(* IEC 61131-3 sources: AXOpen/src/components.dukane.welders/ctrl/src/Axo_IQ_SeriesWelder (part 3) *)

            array_buffer[128] := TO_BYTE(SHR(TO_DWORD(buf2.PressPostWeld.StaticHoldTime), UINT#24));
            array_buffer[129] := TO_BYTE(SHR(TO_DWORD(buf2.PressPostWeld.StaticHoldTime), UINT#16));
            array_buffer[130] := TO_BYTE(SHR(TO_DWORD(buf2.PressPostWeld.StaticHoldTime),  UINT#8));
            array_buffer[131] := TO_BYTE(     TO_DWORD(buf2.PressPostWeld.StaticHoldTime));

            array_buffer[132] := TO_BYTE(SHR(TO_DWORD(buf2.PressPostWeld.AfterburstAmplitude), UINT#24));
            array_buffer[133] := TO_BYTE(SHR(TO_DWORD(buf2.PressPostWeld.AfterburstAmplitude), UINT#16));
            array_buffer[134] := TO_BYTE(SHR(TO_DWORD(buf2.PressPostWeld.AfterburstAmplitude),  UINT#8));
            array_buffer[135] := TO_BYTE(     TO_DWORD(buf2.PressPostWeld.AfterburstAmplitude));

        END_METHOD

        METHOD PRIVATE buf3_TO_ByteArray
            VAR_IN_OUT
                buf3 : Axo_IQ_SeriesWelder_data3_180bytes;
                array_buffer : ARRAY[0..253] OF BYTE;
            END_VAR

            // ---- TriggerTime.Enable bits → bytes 0..3 ----
            array_buffer[ 0].%X0 := buf3.TriggerTime.Enable._0;
            array_buffer[ 0].%X1 := buf3.TriggerTime.Enable._1;
            array_buffer[ 0].%X2 := buf3.TriggerTime.Enable._2;
            array_buffer[ 0].%X3 := buf3.TriggerTime.Enable._3;
            array_buffer[ 0].%X4 := buf3.TriggerTime.Enable._4;
            array_buffer[ 0].%X5 := buf3.TriggerTime.Enable._5;
            array_buffer[ 0].%X6 := buf3.TriggerTime.Enable._6;
            array_buffer[ 0].%X7 := buf3.TriggerTime.Enable._7;

            array_buffer[ 1].%X0 := buf3.TriggerTime.Enable._8;
            array_buffer[ 1].%X1 := buf3.TriggerTime.Enable._9;
            array_buffer[ 1].%X2 := buf3.TriggerTime.Enable._10;
            array_buffer[ 1].%X3 := buf3.TriggerTime.Enable._11;
            array_buffer[ 1].%X4 := buf3.TriggerTime.Enable._12;
            array_buffer[ 1].%X5 := buf3.TriggerTime.Enable._13;
            array_buffer[ 1].%X6 := buf3.TriggerTime.Enable._14;
            array_buffer[ 1].%X7 := buf3.TriggerTime.Enable._15;

            array_buffer[ 2].%X0 := buf3.TriggerTime.Enable._16;
            array_buffer[ 2].%X1 := buf3.TriggerTime.Enable._17;
            array_buffer[ 2].%X2 := buf3.TriggerTime.Enable._18;
            array_buffer[ 2].%X3 := buf3.TriggerTime.Enable._19;
            array_buffer[ 2].%X4 := buf3.TriggerTime.Enable._20;
            array_buffer[ 2].%X5 := buf3.TriggerTime.Enable._21;
            array_buffer[ 2].%X6 := buf3.TriggerTime.Enable._22;
            array_buffer[ 2].%X7 := buf3.TriggerTime.Enable._23;

            array_buffer[ 3].%X0 := buf3.TriggerTime.Enable.LowerBad_1;
            array_buffer[ 3].%X1 := buf3.TriggerTime.Enable.LowerSuspect_1;
            array_buffer[ 3].%X2 := buf3.TriggerTime.Enable.UpperSuspect_1;
            array_buffer[ 3].%X3 := buf3.TriggerTime.Enable.UpperBad_1;
            array_buffer[ 3].%X4 := buf3.TriggerTime.Enable.Display_1;
            array_buffer[ 3].%X5 := buf3.TriggerTime.Enable._29;
            array_buffer[ 3].%X6 := buf3.TriggerTime.Enable._30;
            array_buffer[ 3].%X7 := buf3.TriggerTime.Enable._31;

            // ---- TriggerTime (DINTs) → bytes 4..19 ----
            array_buffer[ 4] := TO_BYTE(SHR(TO_DWORD(buf3.TriggerTime.LowerBad), UINT#24));
            array_buffer[ 5] := TO_BYTE(SHR(TO_DWORD(buf3.TriggerTime.LowerBad), UINT#16));
            array_buffer[ 6] := TO_BYTE(SHR(TO_DWORD(buf3.TriggerTime.LowerBad),  UINT#8));
            array_buffer[ 7] := TO_BYTE(     TO_DWORD(buf3.TriggerTime.LowerBad));

            array_buffer[ 8] := TO_BYTE(SHR(TO_DWORD(buf3.TriggerTime.LowerSuspect), UINT#24));
            array_buffer[ 9] := TO_BYTE(SHR(TO_DWORD(buf3.TriggerTime.LowerSuspect), UINT#16));
            array_buffer[10] := TO_BYTE(SHR(TO_DWORD(buf3.TriggerTime.LowerSuspect),  UINT#8));
            array_buffer[11] := TO_BYTE(     TO_DWORD(buf3.TriggerTime.LowerSuspect));

            array_buffer[12] := TO_BYTE(SHR(TO_DWORD(buf3.TriggerTime.UpperSuspect), UINT#24));
            array_buffer[13] := TO_BYTE(SHR(TO_DWORD(buf3.TriggerTime.UpperSuspect), UINT#16));
            array_buffer[14] := TO_BYTE(SHR(TO_DWORD(buf3.TriggerTime.UpperSuspect),  UINT#8));
            array_buffer[15] := TO_BYTE(     TO_DWORD(buf3.TriggerTime.UpperSuspect));

            array_buffer[16] := TO_BYTE(SHR(TO_DWORD(buf3.TriggerTime.UpperBad), UINT#24));
            array_buffer[17] := TO_BYTE(SHR(TO_DWORD(buf3.TriggerTime.UpperBad), UINT#16));
            array_buffer[18] := TO_BYTE(SHR(TO_DWORD(buf3.TriggerTime.UpperBad),  UINT#8));
            array_buffer[19] := TO_BYTE(     TO_DWORD(buf3.TriggerTime.UpperBad));

            // ---- TriggerPosition.Enable bits → bytes 20..23 ----
            array_buffer[20].%X0 := buf3.TriggerPosition.Enable._0;
            array_buffer[20].%X1 := buf3.TriggerPosition.Enable._1;
            array_buffer[20].%X2 := buf3.TriggerPosition.Enable._2;
            array_buffer[20].%X3 := buf3.TriggerPosition.Enable._3;
            array_buffer[20].%X4 := buf3.TriggerPosition.Enable._4;
            array_buffer[20].%X5 := buf3.TriggerPosition.Enable._5;
            array_buffer[20].%X6 := buf3.TriggerPosition.Enable._6;
            array_buffer[20].%X7 := buf3.TriggerPosition.Enable._7;

            array_buffer[21].%X0 := buf3.TriggerPosition.Enable._8;
            array_buffer[21].%X1 := buf3.TriggerPosition.Enable._9;
            array_buffer[21].%X2 := buf3.TriggerPosition.Enable._10;
            array_buffer[21].%X3 := buf3.TriggerPosition.Enable._11;
            array_buffer[21].%X4 := buf3.TriggerPosition.Enable._12;
            array_buffer[21].%X5 := buf3.TriggerPosition.Enable._13;
            array_buffer[21].%X6 := buf3.TriggerPosition.Enable._14;
            array_buffer[21].%X7 := buf3.TriggerPosition.Enable._15;

            array_buffer[22].%X0 := buf3.TriggerPosition.Enable._16;
            array_buffer[22].%X1 := buf3.TriggerPosition.Enable._17;
            array_buffer[22].%X2 := buf3.TriggerPosition.Enable._18;
            array_buffer[22].%X3 := buf3.TriggerPosition.Enable._19;
            array_buffer[22].%X4 := buf3.TriggerPosition.Enable._20;
            array_buffer[22].%X5 := buf3.TriggerPosition.Enable._21;
            array_buffer[22].%X6 := buf3.TriggerPosition.Enable._22;
            array_buffer[22].%X7 := buf3.TriggerPosition.Enable._23;

            array_buffer[23].%X0 := buf3.TriggerPosition.Enable.LowerBad_1;
            array_buffer[23].%X1 := buf3.TriggerPosition.Enable.LowerSuspect_1;
            array_buffer[23].%X2 := buf3.TriggerPosition.Enable.UpperSuspect_1;
            array_buffer[23].%X3 := buf3.TriggerPosition.Enable.UpperBad_1;
            array_buffer[23].%X4 := buf3.TriggerPosition.Enable.Display_1;
            array_buffer[23].%X5 := buf3.TriggerPosition.Enable._29;
            array_buffer[23].%X6 := buf3.TriggerPosition.Enable._30;
            array_buffer[23].%X7 := buf3.TriggerPosition.Enable._31;

            // ---- TriggerPosition (DINTs) → bytes 24..39 ----
            array_buffer[24] := TO_BYTE(SHR(TO_DWORD(buf3.TriggerPosition.LowerBad), UINT#24));
            array_buffer[25] := TO_BYTE(SHR(TO_DWORD(buf3.TriggerPosition.LowerBad), UINT#16));
            array_buffer[26] := TO_BYTE(SHR(TO_DWORD(buf3.TriggerPosition.LowerBad),  UINT#8));
            array_buffer[27] := TO_BYTE(     TO_DWORD(buf3.TriggerPosition.LowerBad));

            array_buffer[28] := TO_BYTE(SHR(TO_DWORD(buf3.TriggerPosition.LowerSuspect), UINT#24));
            array_buffer[29] := TO_BYTE(SHR(TO_DWORD(buf3.TriggerPosition.LowerSuspect), UINT#16));
            array_buffer[30] := TO_BYTE(SHR(TO_DWORD(buf3.TriggerPosition.LowerSuspect),  UINT#8));
            array_buffer[31] := TO_BYTE(     TO_DWORD(buf3.TriggerPosition.LowerSuspect));

            array_buffer[32] := TO_BYTE(SHR(TO_DWORD(buf3.TriggerPosition.UpperSuspect), UINT#24));
            array_buffer[33] := TO_BYTE(SHR(TO_DWORD(buf3.TriggerPosition.UpperSuspect), UINT#16));
            array_buffer[34] := TO_BYTE(SHR(TO_DWORD(buf3.TriggerPosition.UpperSuspect),  UINT#8));
            array_buffer[35] := TO_BYTE(     TO_DWORD(buf3.TriggerPosition.UpperSuspect));

            array_buffer[36] := TO_BYTE(SHR(TO_DWORD(buf3.TriggerPosition.UpperBad), UINT#24));
            array_buffer[37] := TO_BYTE(SHR(TO_DWORD(buf3.TriggerPosition.UpperBad), UINT#16));
            array_buffer[38] := TO_BYTE(SHR(TO_DWORD(buf3.TriggerPosition.UpperBad),  UINT#8));
            array_buffer[39] := TO_BYTE(     TO_DWORD(buf3.TriggerPosition.UpperBad));

            // ---- TriggerDelayTime.Enable bits → bytes 40..43 ----
            array_buffer[40].%X0 := buf3.TriggerDelayTime.Enable._0;
            array_buffer[40].%X1 := buf3.TriggerDelayTime.Enable._1;
            array_buffer[40].%X2 := buf3.TriggerDelayTime.Enable._2;
            array_buffer[40].%X3 := buf3.TriggerDelayTime.Enable._3;
            array_buffer[40].%X4 := buf3.TriggerDelayTime.Enable._4;
            array_buffer[40].%X5 := buf3.TriggerDelayTime.Enable._5;
            array_buffer[40].%X6 := buf3.TriggerDelayTime.Enable._6;
            array_buffer[40].%X7 := buf3.TriggerDelayTime.Enable._7;

            array_buffer[41].%X0 := buf3.TriggerDelayTime.Enable._8;
            array_buffer[41].%X1 := buf3.TriggerDelayTime.Enable._9;
            array_buffer[41].%X2 := buf3.TriggerDelayTime.Enable._10;
            array_buffer[41].%X3 := buf3.TriggerDelayTime.Enable._11;
            array_buffer[41].%X4 := buf3.TriggerDelayTime.Enable._12;
            array_buffer[41].%X5 := buf3.TriggerDelayTime.Enable._13;
            array_buffer[41].%X6 := buf3.TriggerDelayTime.Enable._14;
            array_buffer[41].%X7 := buf3.TriggerDelayTime.Enable._15;

            array_buffer[42].%X0 := buf3.TriggerDelayTime.Enable._16;
            array_buffer[42].%X1 := buf3.TriggerDelayTime.Enable._17;
            array_buffer[42].%X2 := buf3.TriggerDelayTime.Enable._18;
            array_buffer[42].%X3 := buf3.TriggerDelayTime.Enable._19;
            array_buffer[42].%X4 := buf3.TriggerDelayTime.Enable._20;
            array_buffer[42].%X5 := buf3.TriggerDelayTime.Enable._21;
            array_buffer[42].%X6 := buf3.TriggerDelayTime.Enable._22;
            array_buffer[42].%X7 := buf3.TriggerDelayTime.Enable._23;

            array_buffer[43].%X0 := buf3.TriggerDelayTime.Enable.LowerBad_1;
            array_buffer[43].%X1 := buf3.TriggerDelayTime.Enable.LowerSuspect_1;
            array_buffer[43].%X2 := buf3.TriggerDelayTime.Enable.UpperSuspect_1;
            array_buffer[43].%X3 := buf3.TriggerDelayTime.Enable.UpperBad_1;
            array_buffer[43].%X4 := buf3.TriggerDelayTime.Enable.Display_1;
            array_buffer[43].%X5 := buf3.TriggerDelayTime.Enable._29;
            array_buffer[43].%X6 := buf3.TriggerDelayTime.Enable._30;
            array_buffer[43].%X7 := buf3.TriggerDelayTime.Enable._31;

            // ---- TriggerDelayTime (DINTs) → bytes 44..59 ----
            array_buffer[44] := TO_BYTE(SHR(TO_DWORD(buf3.TriggerDelayTime.LowerBad), UINT#24));
            array_buffer[45] := TO_BYTE(SHR(TO_DWORD(buf3.TriggerDelayTime.LowerBad), UINT#16));
            array_buffer[46] := TO_BYTE(SHR(TO_DWORD(buf3.TriggerDelayTime.LowerBad),  UINT#8));
            array_buffer[47] := TO_BYTE(     TO_DWORD(buf3.TriggerDelayTime.LowerBad));

            array_buffer[48] := TO_BYTE(SHR(TO_DWORD(buf3.TriggerDelayTime.LowerSuspect), UINT#24));
            array_buffer[49] := TO_BYTE(SHR(TO_DWORD(buf3.TriggerDelayTime.LowerSuspect), UINT#16));
            array_buffer[50] := TO_BYTE(SHR(TO_DWORD(buf3.TriggerDelayTime.LowerSuspect),  UINT#8));
            array_buffer[51] := TO_BYTE(     TO_DWORD(buf3.TriggerDelayTime.LowerSuspect));

            array_buffer[52] := TO_BYTE(SHR(TO_DWORD(buf3.TriggerDelayTime.UpperSuspect), UINT#24));
            array_buffer[53] := TO_BYTE(SHR(TO_DWORD(buf3.TriggerDelayTime.UpperSuspect), UINT#16));
            array_buffer[54] := TO_BYTE(SHR(TO_DWORD(buf3.TriggerDelayTime.UpperSuspect),  UINT#8));
            array_buffer[55] := TO_BYTE(     TO_DWORD(buf3.TriggerDelayTime.UpperSuspect));

            array_buffer[56] := TO_BYTE(SHR(TO_DWORD(buf3.TriggerDelayTime.UpperBad), UINT#24));
            array_buffer[57] := TO_BYTE(SHR(TO_DWORD(buf3.TriggerDelayTime.UpperBad), UINT#16));
            array_buffer[58] := TO_BYTE(SHR(TO_DWORD(buf3.TriggerDelayTime.UpperBad),  UINT#8));
            array_buffer[59] := TO_BYTE(     TO_DWORD(buf3.TriggerDelayTime.UpperBad));

            // ---- TriggerDelayDistance.Enable bits → bytes 60..63 ----
            array_buffer[60].%X0 := buf3.TriggerDelayDistance.Enable._0;
            array_buffer[60].%X1 := buf3.TriggerDelayDistance.Enable._1;
            array_buffer[60].%X2 := buf3.TriggerDelayDistance.Enable._2;
            array_buffer[60].%X3 := buf3.TriggerDelayDistance.Enable._3;
            array_buffer[60].%X4 := buf3.TriggerDelayDistance.Enable._4;
            array_buffer[60].%X5 := buf3.TriggerDelayDistance.Enable._5;
            array_buffer[60].%X6 := buf3.TriggerDelayDistance.Enable._6;
            array_buffer[60].%X7 := buf3.TriggerDelayDistance.Enable._7;

            array_buffer[61].%X0 := buf3.TriggerDelayDistance.Enable._8;
            array_buffer[61].%X1 := buf3.TriggerDelayDistance.Enable._9;
            array_buffer[61].%X2 := buf3.TriggerDelayDistance.Enable._10;
            array_buffer[61].%X3 := buf3.TriggerDelayDistance.Enable._11;
            array_buffer[61].%X4 := buf3.TriggerDelayDistance.Enable._12;
            array_buffer[61].%X5 := buf3.TriggerDelayDistance.Enable._13;
            array_buffer[61].%X6 := buf3.TriggerDelayDistance.Enable._14;
            array_buffer[61].%X7 := buf3.TriggerDelayDistance.Enable._15;

            array_buffer[62].%X0 := buf3.TriggerDelayDistance.Enable._16;
            array_buffer[62].%X1 := buf3.TriggerDelayDistance.Enable._17;
            array_buffer[62].%X2 := buf3.TriggerDelayDistance.Enable._18;
            array_buffer[62].%X3 := buf3.TriggerDelayDistance.Enable._19;
            array_buffer[62].%X4 := buf3.TriggerDelayDistance.Enable._20;
            array_buffer[62].%X5 := buf3.TriggerDelayDistance.Enable._21;
            array_buffer[62].%X6 := buf3.TriggerDelayDistance.Enable._22;
            array_buffer[62].%X7 := buf3.TriggerDelayDistance.Enable._23;

            array_buffer[63].%X0 := buf3.TriggerDelayDistance.Enable.LowerBad_1;
            array_buffer[63].%X1 := buf3.TriggerDelayDistance.Enable.LowerSuspect_1;
            array_buffer[63].%X2 := buf3.TriggerDelayDistance.Enable.UpperSuspect_1;
            array_buffer[63].%X3 := buf3.TriggerDelayDistance.Enable.UpperBad_1;
            array_buffer[63].%X4 := buf3.TriggerDelayDistance.Enable.Display_1;
            array_buffer[63].%X5 := buf3.TriggerDelayDistance.Enable._29;
            array_buffer[63].%X6 := buf3.TriggerDelayDistance.Enable._30;
            array_buffer[63].%X7 := buf3.TriggerDelayDistance.Enable._31;

            // ---- TriggerDelayDistance (DINTs) → bytes 64..79 ----
            array_buffer[64] := TO_BYTE(SHR(TO_DWORD(buf3.TriggerDelayDistance.LowerBad), UINT#24));
            array_buffer[65] := TO_BYTE(SHR(TO_DWORD(buf3.TriggerDelayDistance.LowerBad), UINT#16));
            array_buffer[66] := TO_BYTE(SHR(TO_DWORD(buf3.TriggerDelayDistance.LowerBad),  UINT#8));
            array_buffer[67] := TO_BYTE(     TO_DWORD(buf3.TriggerDelayDistance.LowerBad));

            array_buffer[68] := TO_BYTE(SHR(TO_DWORD(buf3.TriggerDelayDistance.LowerSuspect), UINT#24));
            array_buffer[69] := TO_BYTE(SHR(TO_DWORD(buf3.TriggerDelayDistance.LowerSuspect), UINT#16));
            array_buffer[70] := TO_BYTE(SHR(TO_DWORD(buf3.TriggerDelayDistance.LowerSuspect),  UINT#8));
            array_buffer[71] := TO_BYTE(     TO_DWORD(buf3.TriggerDelayDistance.LowerSuspect));

            array_buffer[72] := TO_BYTE(SHR(TO_DWORD(buf3.TriggerDelayDistance.UpperSuspect), UINT#24));
            array_buffer[73] := TO_BYTE(SHR(TO_DWORD(buf3.TriggerDelayDistance.UpperSuspect), UINT#16));
            array_buffer[74] := TO_BYTE(SHR(TO_DWORD(buf3.TriggerDelayDistance.UpperSuspect),  UINT#8));
            array_buffer[75] := TO_BYTE(     TO_DWORD(buf3.TriggerDelayDistance.UpperSuspect));

            array_buffer[76] := TO_BYTE(SHR(TO_DWORD(buf3.TriggerDelayDistance.UpperBad), UINT#24));
            array_buffer[77] := TO_BYTE(SHR(TO_DWORD(buf3.TriggerDelayDistance.UpperBad), UINT#16));
            array_buffer[78] := TO_BYTE(SHR(TO_DWORD(buf3.TriggerDelayDistance.UpperBad),  UINT#8));
            array_buffer[79] := TO_BYTE(     TO_DWORD(buf3.TriggerDelayDistance.UpperBad));

            // ---- Weld1Distance.Enable bits → bytes 80..83 ----
            array_buffer[80].%X0 := buf3.Weld1Distance.Enable._0;
            array_buffer[80].%X1 := buf3.Weld1Distance.Enable._1;
            array_buffer[80].%X2 := buf3.Weld1Distance.Enable._2;
            array_buffer[80].%X3 := buf3.Weld1Distance.Enable._3;
            array_buffer[80].%X4 := buf3.Weld1Distance.Enable._4;
            array_buffer[80].%X5 := buf3.Weld1Distance.Enable._5;
            array_buffer[80].%X6 := buf3.Weld1Distance.Enable._6;
            array_buffer[80].%X7 := buf3.Weld1Distance.Enable._7;

            array_buffer[81].%X0 := buf3.Weld1Distance.Enable._8;
            array_buffer[81].%X1 := buf3.Weld1Distance.Enable._9;
            array_buffer[81].%X2 := buf3.Weld1Distance.Enable._10;
            array_buffer[81].%X3 := buf3.Weld1Distance.Enable._11;
            array_buffer[81].%X4 := buf3.Weld1Distance.Enable._12;
            array_buffer[81].%X5 := buf3.Weld1Distance.Enable._13;
            array_buffer[81].%X6 := buf3.Weld1Distance.Enable._14;
            array_buffer[81].%X7 := buf3.Weld1Distance.Enable._15;

            array_buffer[82].%X0 := buf3.Weld1Distance.Enable._16;
            array_buffer[82].%X1 := buf3.Weld1Distance.Enable._17;
            array_buffer[82].%X2 := buf3.Weld1Distance.Enable._18;
            array_buffer[82].%X3 := buf3.Weld1Distance.Enable._19;
            array_buffer[82].%X4 := buf3.Weld1Distance.Enable._20;
            array_buffer[82].%X5 := buf3.Weld1Distance.Enable._21;
            array_buffer[82].%X6 := buf3.Weld1Distance.Enable._22;
            array_buffer[82].%X7 := buf3.Weld1Distance.Enable._23;

            array_buffer[83].%X0 := buf3.Weld1Distance.Enable.LowerBad_1;
            array_buffer[83].%X1 := buf3.Weld1Distance.Enable.LowerSuspect_1;
            array_buffer[83].%X2 := buf3.Weld1Distance.Enable.UpperSuspect_1;
            array_buffer[83].%X3 := buf3.Weld1Distance.Enable.UpperBad_1;
            array_buffer[83].%X4 := buf3.Weld1Distance.Enable.Display_1;
            array_buffer[83].%X5 := buf3.Weld1Distance.Enable._29;
            array_buffer[83].%X6 := buf3.Weld1Distance.Enable._30;
            array_buffer[83].%X7 := buf3.Weld1Distance.Enable._31;

            // ---- Weld1Distance (DINTs) → bytes 84..99 ----
            array_buffer[84] := TO_BYTE(SHR(TO_DWORD(buf3.Weld1Distance.LowerBad), UINT#24));
            array_buffer[85] := TO_BYTE(SHR(TO_DWORD(buf3.Weld1Distance.LowerBad), UINT#16));
            array_buffer[86] := TO_BYTE(SHR(TO_DWORD(buf3.Weld1Distance.LowerBad),  UINT#8));
            array_buffer[87] := TO_BYTE(     TO_DWORD(buf3.Weld1Distance.LowerBad));

            array_buffer[88] := TO_BYTE(SHR(TO_DWORD(buf3.Weld1Distance.LowerSuspect), UINT#24));
            array_buffer[89] := TO_BYTE(SHR(TO_DWORD(buf3.Weld1Distance.LowerSuspect), UINT#16));
            array_buffer[90] := TO_BYTE(SHR(TO_DWORD(buf3.Weld1Distance.LowerSuspect),  UINT#8));
            array_buffer[91] := TO_BYTE(     TO_DWORD(buf3.Weld1Distance.LowerSuspect));

            array_buffer[92] := TO_BYTE(SHR(TO_DWORD(buf3.Weld1Distance.UpperSuspect), UINT#24));
            array_buffer[93] := TO_BYTE(SHR(TO_DWORD(buf3.Weld1Distance.UpperSuspect), UINT#16));
            array_buffer[94] := TO_BYTE(SHR(TO_DWORD(buf3.Weld1Distance.UpperSuspect),  UINT#8));
            array_buffer[95] := TO_BYTE(     TO_DWORD(buf3.Weld1Distance.UpperSuspect));

            array_buffer[96] := TO_BYTE(SHR(TO_DWORD(buf3.Weld1Distance.UpperBad), UINT#24));
            array_buffer[97] := TO_BYTE(SHR(TO_DWORD(buf3.Weld1Distance.UpperBad), UINT#16));
            array_buffer[98] := TO_BYTE(SHR(TO_DWORD(buf3.Weld1Distance.UpperBad),  UINT#8));
            array_buffer[99] := TO_BYTE(     TO_DWORD(buf3.Weld1Distance.UpperBad));

            // ---- Weld1Position.Enable bits → bytes 100..103 ----
            array_buffer[100].%X0 := buf3.Weld1Position.Enable._0;
            array_buffer[100].%X1 := buf3.Weld1Position.Enable._1;
            array_buffer[100].%X2 := buf3.Weld1Position.Enable._2;
            array_buffer[100].%X3 := buf3.Weld1Position.Enable._3;
            array_buffer[100].%X4 := buf3.Weld1Position.Enable._4;
            array_buffer[100].%X5 := buf3.Weld1Position.Enable._5;
            array_buffer[100].%X6 := buf3.Weld1Position.Enable._6;
            array_buffer[100].%X7 := buf3.Weld1Position.Enable._7;

            array_buffer[101].%X0 := buf3.Weld1Position.Enable._8;
            array_buffer[101].%X1 := buf3.Weld1Position.Enable._9;
            array_buffer[101].%X2 := buf3.Weld1Position.Enable._10;
            array_buffer[101].%X3 := buf3.Weld1Position.Enable._11;
            array_buffer[101].%X4 := buf3.Weld1Position.Enable._12;
            array_buffer[101].%X5 := buf3.Weld1Position.Enable._13;
            array_buffer[101].%X6 := buf3.Weld1Position.Enable._14;
            array_buffer[101].%X7 := buf3.Weld1Position.Enable._15;

            array_buffer[102].%X0 := buf3.Weld1Position.Enable._16;
            array_buffer[102].%X1 := buf3.Weld1Position.Enable._17;
            array_buffer[102].%X2 := buf3.Weld1Position.Enable._18;
            array_buffer[102].%X3 := buf3.Weld1Position.Enable._19;
            array_buffer[102].%X4 := buf3.Weld1Position.Enable._20;
            array_buffer[102].%X5 := buf3.Weld1Position.Enable._21;
            array_buffer[102].%X6 := buf3.Weld1Position.Enable._22;
            array_buffer[102].%X7 := buf3.Weld1Position.Enable._23;

            array_buffer[103].%X0 := buf3.Weld1Position.Enable.LowerBad_1;
            array_buffer[103].%X1 := buf3.Weld1Position.Enable.LowerSuspect_1;
            array_buffer[103].%X2 := buf3.Weld1Position.Enable.UpperSuspect_1;
            array_buffer[103].%X3 := buf3.Weld1Position.Enable.UpperBad_1;
            array_buffer[103].%X4 := buf3.Weld1Position.Enable.Display_1;
            array_buffer[103].%X5 := buf3.Weld1Position.Enable._29;
            array_buffer[103].%X6 := buf3.Weld1Position.Enable._30;
            array_buffer[103].%X7 := buf3.Weld1Position.Enable._31;

            // ---- Weld1Position (DINTs) → bytes 104..119 ----
            array_buffer[104] := TO_BYTE(SHR(TO_DWORD(buf3.Weld1Position.LowerBad), UINT#24));
            array_buffer[105] := TO_BYTE(SHR(TO_DWORD(buf3.Weld1Position.LowerBad), UINT#16));
            array_buffer[106] := TO_BYTE(SHR(TO_DWORD(buf3.Weld1Position.LowerBad),  UINT#8));
            array_buffer[107] := TO_BYTE(     TO_DWORD(buf3.Weld1Position.LowerBad));

            array_buffer[108] := TO_BYTE(SHR(TO_DWORD(buf3.Weld1Position.LowerSuspect), UINT#24));
            array_buffer[109] := TO_BYTE(SHR(TO_DWORD(buf3.Weld1Position.LowerSuspect), UINT#16));
            array_buffer[110] := TO_BYTE(SHR(TO_DWORD(buf3.Weld1Position.LowerSuspect),  UINT#8));
            array_buffer[111] := TO_BYTE(     TO_DWORD(buf3.Weld1Position.LowerSuspect));

            array_buffer[112] := TO_BYTE(SHR(TO_DWORD(buf3.Weld1Position.UpperSuspect), UINT#24));
            array_buffer[113] := TO_BYTE(SHR(TO_DWORD(buf3.Weld1Position.UpperSuspect), UINT#16));
            array_buffer[114] := TO_BYTE(SHR(TO_DWORD(buf3.Weld1Position.UpperSuspect),  UINT#8));
            array_buffer[115] := TO_BYTE(     TO_DWORD(buf3.Weld1Position.UpperSuspect));

            array_buffer[116] := TO_BYTE(SHR(TO_DWORD(buf3.Weld1Position.UpperBad), UINT#24));
            array_buffer[117] := TO_BYTE(SHR(TO_DWORD(buf3.Weld1Position.UpperBad), UINT#16));
            array_buffer[118] := TO_BYTE(SHR(TO_DWORD(buf3.Weld1Position.UpperBad),  UINT#8));
            array_buffer[119] := TO_BYTE(     TO_DWORD(buf3.Weld1Position.UpperBad));

            // ---- Weld2Time.Enable bits → bytes 120..123 ----
            array_buffer[120].%X0 := buf3.Weld2Time.Enable._0;
            array_buffer[120].%X1 := buf3.Weld2Time.Enable._1;
            array_buffer[120].%X2 := buf3.Weld2Time.Enable._2;
            array_buffer[120].%X3 := buf3.Weld2Time.Enable._3;
            array_buffer[120].%X4 := buf3.Weld2Time.Enable._4;
            array_buffer[120].%X5 := buf3.Weld2Time.Enable._5;
            array_buffer[120].%X6 := buf3.Weld2Time.Enable._6;
            array_buffer[120].%X7 := buf3.Weld2Time.Enable._7;

            array_buffer[121].%X0 := buf3.Weld2Time.Enable._8;
            array_buffer[121].%X1 := buf3.Weld2Time.Enable._9;
            array_buffer[121].%X2 := buf3.Weld2Time.Enable._10;
            array_buffer[121].%X3 := buf3.Weld2Time.Enable._11;
            array_buffer[121].%X4 := buf3.Weld2Time.Enable._12;
            array_buffer[121].%X5 := buf3.Weld2Time.Enable._13;
            array_buffer[121].%X6 := buf3.Weld2Time.Enable._14;
            array_buffer[121].%X7 := buf3.Weld2Time.Enable._15;

            array_buffer[122].%X0 := buf3.Weld2Time.Enable._16;
            array_buffer[122].%X1 := buf3.Weld2Time.Enable._17;
            array_buffer[122].%X2 := buf3.Weld2Time.Enable._18;
            array_buffer[122].%X3 := buf3.Weld2Time.Enable._19;
            array_buffer[122].%X4 := buf3.Weld2Time.Enable._20;
            array_buffer[122].%X5 := buf3.Weld2Time.Enable._21;
            array_buffer[122].%X6 := buf3.Weld2Time.Enable._22;
            array_buffer[122].%X7 := buf3.Weld2Time.Enable._23;

            array_buffer[123].%X0 := buf3.Weld2Time.Enable.LowerBad_1;
            array_buffer[123].%X1 := buf3.Weld2Time.Enable.LowerSuspect_1;
            array_buffer[123].%X2 := buf3.Weld2Time.Enable.UpperSuspect_1;
            array_buffer[123].%X3 := buf3.Weld2Time.Enable.UpperBad_1;
            array_buffer[123].%X4 := buf3.Weld2Time.Enable.Display_1;
            array_buffer[123].%X5 := buf3.Weld2Time.Enable._29;
            array_buffer[123].%X6 := buf3.Weld2Time.Enable._30;
            array_buffer[123].%X7 := buf3.Weld2Time.Enable._31;

            // ---- Weld2Time (DINTs) → bytes 124..139 ----
            array_buffer[124] := TO_BYTE(SHR(TO_DWORD(buf3.Weld2Time.LowerBad), UINT#24));
            array_buffer[125] := TO_BYTE(SHR(TO_DWORD(buf3.Weld2Time.LowerBad), UINT#16));
            array_buffer[126] := TO_BYTE(SHR(TO_DWORD(buf3.Weld2Time.LowerBad),  UINT#8));
            array_buffer[127] := TO_BYTE(     TO_DWORD(buf3.Weld2Time.LowerBad));

            array_buffer[128] := TO_BYTE(SHR(TO_DWORD(buf3.Weld2Time.LowerSuspect), UINT#24));
            array_buffer[129] := TO_BYTE(SHR(TO_DWORD(buf3.Weld2Time.LowerSuspect), UINT#16));
            array_buffer[130] := TO_BYTE(SHR(TO_DWORD(buf3.Weld2Time.LowerSuspect),  UINT#8));
            array_buffer[131] := TO_BYTE(     TO_DWORD(buf3.Weld2Time.LowerSuspect));

            array_buffer[132] := TO_BYTE(SHR(TO_DWORD(buf3.Weld2Time.UpperSuspect), UINT#24));
            array_buffer[133] := TO_BYTE(SHR(TO_DWORD(buf3.Weld2Time.UpperSuspect), UINT#16));
            array_buffer[134] := TO_BYTE(SHR(TO_DWORD(buf3.Weld2Time.UpperSuspect),  UINT#8));
            array_buffer[135] := TO_BYTE(     TO_DWORD(buf3.Weld2Time.UpperSuspect));

            array_buffer[136] := TO_BYTE(SHR(TO_DWORD(buf3.Weld2Time.UpperBad), UINT#24));
            array_buffer[137] := TO_BYTE(SHR(TO_DWORD(buf3.Weld2Time.UpperBad), UINT#16));
            array_buffer[138] := TO_BYTE(SHR(TO_DWORD(buf3.Weld2Time.UpperBad),  UINT#8));
            array_buffer[139] := TO_BYTE(     TO_DWORD(buf3.Weld2Time.UpperBad));

            // ---- Weld2Energy.Enable bits → bytes 140..143 ----
            array_buffer[140].%X0 := buf3.Weld2Energy.Enable._0;
            array_buffer[140].%X1 := buf3.Weld2Energy.Enable._1;
            array_buffer[140].%X2 := buf3.Weld2Energy.Enable._2;
            array_buffer[140].%X3 := buf3.Weld2Energy.Enable._3;
            array_buffer[140].%X4 := buf3.Weld2Energy.Enable._4;
            array_buffer[140].%X5 := buf3.Weld2Energy.Enable._5;
            array_buffer[140].%X6 := buf3.Weld2Energy.Enable._6;
            array_buffer[140].%X7 := buf3.Weld2Energy.Enable._7;

            array_buffer[141].%X0 := buf3.Weld2Energy.Enable._8;
            array_buffer[141].%X1 := buf3.Weld2Energy.Enable._9;
            array_buffer[141].%X2 := buf3.Weld2Energy.Enable._10;
            array_buffer[141].%X3 := buf3.Weld2Energy.Enable._11;
            array_buffer[141].%X4 := buf3.Weld2Energy.Enable._12;
            array_buffer[141].%X5 := buf3.Weld2Energy.Enable._13;
            array_buffer[141].%X6 := buf3.Weld2Energy.Enable._14;
            array_buffer[141].%X7 := buf3.Weld2Energy.Enable._15;

            array_buffer[142].%X0 := buf3.Weld2Energy.Enable._16;
            array_buffer[142].%X1 := buf3.Weld2Energy.Enable._17;
            array_buffer[142].%X2 := buf3.Weld2Energy.Enable._18;
            array_buffer[142].%X3 := buf3.Weld2Energy.Enable._19;
            array_buffer[142].%X4 := buf3.Weld2Energy.Enable._20;
            array_buffer[142].%X5 := buf3.Weld2Energy.Enable._21;
            array_buffer[142].%X6 := buf3.Weld2Energy.Enable._22;
            array_buffer[142].%X7 := buf3.Weld2Energy.Enable._23;

            array_buffer[143].%X0 := buf3.Weld2Energy.Enable.LowerBad_1;
            array_buffer[143].%X1 := buf3.Weld2Energy.Enable.LowerSuspect_1;
            array_buffer[143].%X2 := buf3.Weld2Energy.Enable.UpperSuspect_1;
            array_buffer[143].%X3 := buf3.Weld2Energy.Enable.UpperBad_1;
            array_buffer[143].%X4 := buf3.Weld2Energy.Enable.Display_1;
            array_buffer[143].%X5 := buf3.Weld2Energy.Enable._29;
            array_buffer[143].%X6 := buf3.Weld2Energy.Enable._30;
            array_buffer[143].%X7 := buf3.Weld2Energy.Enable._31;

            // ---- Weld2Energy (DINTs) → bytes 144..159 ----
            array_buffer[144] := TO_BYTE(SHR(TO_DWORD(buf3.Weld2Energy.LowerBad), UINT#24));
            array_buffer[145] := TO_BYTE(SHR(TO_DWORD(buf3.Weld2Energy.LowerBad), UINT#16));
            array_buffer[146] := TO_BYTE(SHR(TO_DWORD(buf3.Weld2Energy.LowerBad),  UINT#8));
            array_buffer[147] := TO_BYTE(     TO_DWORD(buf3.Weld2Energy.LowerBad));

            array_buffer[148] := TO_BYTE(SHR(TO_DWORD(buf3.Weld2Energy.LowerSuspect), UINT#24));
            array_buffer[149] := TO_BYTE(SHR(TO_DWORD(buf3.Weld2Energy.LowerSuspect), UINT#16));
            array_buffer[150] := TO_BYTE(SHR(TO_DWORD(buf3.Weld2Energy.LowerSuspect),  UINT#8));
            array_buffer[151] := TO_BYTE(     TO_DWORD(buf3.Weld2Energy.LowerSuspect));

            array_buffer[152] := TO_BYTE(SHR(TO_DWORD(buf3.Weld2Energy.UpperSuspect), UINT#24));
            array_buffer[153] := TO_BYTE(SHR(TO_DWORD(buf3.Weld2Energy.UpperSuspect), UINT#16));
            array_buffer[154] := TO_BYTE(SHR(TO_DWORD(buf3.Weld2Energy.UpperSuspect),  UINT#8));
            array_buffer[155] := TO_BYTE(     TO_DWORD(buf3.Weld2Energy.UpperSuspect));

            array_buffer[156] := TO_BYTE(SHR(TO_DWORD(buf3.Weld2Energy.UpperBad), UINT#24));
            array_buffer[157] := TO_BYTE(SHR(TO_DWORD(buf3.Weld2Energy.UpperBad), UINT#16));
            array_buffer[158] := TO_BYTE(SHR(TO_DWORD(buf3.Weld2Energy.UpperBad),  UINT#8));
            array_buffer[159] := TO_BYTE(     TO_DWORD(buf3.Weld2Energy.UpperBad));

            // ---- Weld2Power.Enable bits → bytes 160..163 ----
            array_buffer[160].%X0 := buf3.Weld2Power.Enable._0;
            array_buffer[160].%X1 := buf3.Weld2Power.Enable._1;
            array_buffer[160].%X2 := buf3.Weld2Power.Enable._2;
            array_buffer[160].%X3 := buf3.Weld2Power.Enable._3;
            array_buffer[160].%X4 := buf3.Weld2Power.Enable._4;
            array_buffer[160].%X5 := buf3.Weld2Power.Enable._5;
            array_buffer[160].%X6 := buf3.Weld2Power.Enable._6;
            array_buffer[160].%X7 := buf3.Weld2Power.Enable._7;

            array_buffer[161].%X0 := buf3.Weld2Power.Enable._8;
            array_buffer[161].%X1 := buf3.Weld2Power.Enable._9;
            array_buffer[161].%X2 := buf3.Weld2Power.Enable._10;
            array_buffer[161].%X3 := buf3.Weld2Power.Enable._11;
            array_buffer[161].%X4 := buf3.Weld2Power.Enable._12;
            array_buffer[161].%X5 := buf3.Weld2Power.Enable._13;
            array_buffer[161].%X6 := buf3.Weld2Power.Enable._14;
            array_buffer[161].%X7 := buf3.Weld2Power.Enable._15;

            array_buffer[162].%X0 := buf3.Weld2Power.Enable._16;
            array_buffer[162].%X1 := buf3.Weld2Power.Enable._17;
            array_buffer[162].%X2 := buf3.Weld2Power.Enable._18;
            array_buffer[162].%X3 := buf3.Weld2Power.Enable._19;
            array_buffer[162].%X4 := buf3.Weld2Power.Enable._20;
            array_buffer[162].%X5 := buf3.Weld2Power.Enable._21;
            array_buffer[162].%X6 := buf3.Weld2Power.Enable._22;
            array_buffer[162].%X7 := buf3.Weld2Power.Enable._23;

            array_buffer[163].%X0 := buf3.Weld2Power.Enable.LowerBad_1;
            array_buffer[163].%X1 := buf3.Weld2Power.Enable.LowerSuspect_1;
            array_buffer[163].%X2 := buf3.Weld2Power.Enable.UpperSuspect_1;
            array_buffer[163].%X3 := buf3.Weld2Power.Enable.UpperBad_1;
            array_buffer[163].%X4 := buf3.Weld2Power.Enable.Display_1;
            array_buffer[163].%X5 := buf3.Weld2Power.Enable._29;
            array_buffer[163].%X6 := buf3.Weld2Power.Enable._30;
            array_buffer[163].%X7 := buf3.Weld2Power.Enable._31;

            // ---- Weld2Power (DINTs) → bytes 164..179 ----
            array_buffer[164] := TO_BYTE(SHR(TO_DWORD(buf3.Weld2Power.LowerBad), UINT#24));
            array_buffer[165] := TO_BYTE(SHR(TO_DWORD(buf3.Weld2Power.LowerBad), UINT#16));
            array_buffer[166] := TO_BYTE(SHR(TO_DWORD(buf3.Weld2Power.LowerBad),  UINT#8));
            array_buffer[167] := TO_BYTE(     TO_DWORD(buf3.Weld2Power.LowerBad));

            array_buffer[168] := TO_BYTE(SHR(TO_DWORD(buf3.Weld2Power.LowerSuspect), UINT#24));
            array_buffer[169] := TO_BYTE(SHR(TO_DWORD(buf3.Weld2Power.LowerSuspect), UINT#16));
            array_buffer[170] := TO_BYTE(SHR(TO_DWORD(buf3.Weld2Power.LowerSuspect),  UINT#8));
            array_buffer[171] := TO_BYTE(     TO_DWORD(buf3.Weld2Power.LowerSuspect));

            array_buffer[172] := TO_BYTE(SHR(TO_DWORD(buf3.Weld2Power.UpperSuspect), UINT#24));
            array_buffer[173] := TO_BYTE(SHR(TO_DWORD(buf3.Weld2Power.UpperSuspect), UINT#16));
            array_buffer[174] := TO_BYTE(SHR(TO_DWORD(buf3.Weld2Power.UpperSuspect),  UINT#8));
            array_buffer[175] := TO_BYTE(     TO_DWORD(buf3.Weld2Power.UpperSuspect));

            array_buffer[176] := TO_BYTE(SHR(TO_DWORD(buf3.Weld2Power.UpperBad), UINT#24));
            array_buffer[177] := TO_BYTE(SHR(TO_DWORD(buf3.Weld2Power.UpperBad), UINT#16));
            array_buffer[178] := TO_BYTE(SHR(TO_DWORD(buf3.Weld2Power.UpperBad),  UINT#8));
            array_buffer[179] := TO_BYTE(     TO_DWORD(buf3.Weld2Power.UpperBad));

        END_METHOD

        METHOD PRIVATE buf4_TO_ByteArray
            VAR_IN_OUT
                buf4 : Axo_IQ_SeriesWelder_data4_200bytes;
                array_buffer : ARRAY[0..253] OF BYTE;
            END_VAR

            // ---- Weld2Distance.Enable bits → bytes 0..3 ----
            array_buffer[ 0].%X0 := buf4.Weld2Distance.Enable._0;
            array_buffer[ 0].%X1 := buf4.Weld2Distance.Enable._1;
            array_buffer[ 0].%X2 := buf4.Weld2Distance.Enable._2;
            array_buffer[ 0].%X3 := buf4.Weld2Distance.Enable._3;
            array_buffer[ 0].%X4 := buf4.Weld2Distance.Enable._4;
            array_buffer[ 0].%X5 := buf4.Weld2Distance.Enable._5;
            array_buffer[ 0].%X6 := buf4.Weld2Distance.Enable._6;
            array_buffer[ 0].%X7 := buf4.Weld2Distance.Enable._7;

            array_buffer[ 1].%X0 := buf4.Weld2Distance.Enable._8;
            array_buffer[ 1].%X1 := buf4.Weld2Distance.Enable._9;
            array_buffer[ 1].%X2 := buf4.Weld2Distance.Enable._10;
            array_buffer[ 1].%X3 := buf4.Weld2Distance.Enable._11;
            array_buffer[ 1].%X4 := buf4.Weld2Distance.Enable._12;
            array_buffer[ 1].%X5 := buf4.Weld2Distance.Enable._13;
            array_buffer[ 1].%X6 := buf4.Weld2Distance.Enable._14;
            array_buffer[ 1].%X7 := buf4.Weld2Distance.Enable._15;

            array_buffer[ 2].%X0 := buf4.Weld2Distance.Enable._16;
            array_buffer[ 2].%X1 := buf4.Weld2Distance.Enable._17;
            array_buffer[ 2].%X2 := buf4.Weld2Distance.Enable._18;
            array_buffer[ 2].%X3 := buf4.Weld2Distance.Enable._19;
            array_buffer[ 2].%X4 := buf4.Weld2Distance.Enable._20;
            array_buffer[ 2].%X5 := buf4.Weld2Distance.Enable._21;
            array_buffer[ 2].%X6 := buf4.Weld2Distance.Enable._22;
            array_buffer[ 2].%X7 := buf4.Weld2Distance.Enable._23;

            array_buffer[ 3].%X0 := buf4.Weld2Distance.Enable.LowerBad_1;
            array_buffer[ 3].%X1 := buf4.Weld2Distance.Enable.LowerSuspect_1;
            array_buffer[ 3].%X2 := buf4.Weld2Distance.Enable.UpperSuspect_1;
            array_buffer[ 3].%X3 := buf4.Weld2Distance.Enable.UpperBad_1;
            array_buffer[ 3].%X4 := buf4.Weld2Distance.Enable.Display_1;
            array_buffer[ 3].%X5 := buf4.Weld2Distance.Enable._29;
            array_buffer[ 3].%X6 := buf4.Weld2Distance.Enable._30;
            array_buffer[ 3].%X7 := buf4.Weld2Distance.Enable._31;

            // ---- Weld2Distance (DINTs) → bytes 4..19 ----
            array_buffer[ 4] := TO_BYTE(SHR(TO_DWORD(buf4.Weld2Distance.LowerBad), UINT#24));
            array_buffer[ 5] := TO_BYTE(SHR(TO_DWORD(buf4.Weld2Distance.LowerBad), UINT#16));
            array_buffer[ 6] := TO_BYTE(SHR(TO_DWORD(buf4.Weld2Distance.LowerBad),  UINT#8));
            array_buffer[ 7] := TO_BYTE(     TO_DWORD(buf4.Weld2Distance.LowerBad));

            array_buffer[ 8] := TO_BYTE(SHR(TO_DWORD(buf4.Weld2Distance.LowerSuspect), UINT#24));
            array_buffer[ 9] := TO_BYTE(SHR(TO_DWORD(buf4.Weld2Distance.LowerSuspect), UINT#16));
            array_buffer[10] := TO_BYTE(SHR(TO_DWORD(buf4.Weld2Distance.LowerSuspect),  UINT#8));
            array_buffer[11] := TO_BYTE(     TO_DWORD(buf4.Weld2Distance.LowerSuspect));

            array_buffer[12] := TO_BYTE(SHR(TO_DWORD(buf4.Weld2Distance.UpperSuspect), UINT#24));
            array_buffer[13] := TO_BYTE(SHR(TO_DWORD(buf4.Weld2Distance.UpperSuspect), UINT#16));
            array_buffer[14] := TO_BYTE(SHR(TO_DWORD(buf4.Weld2Distance.UpperSuspect),  UINT#8));
            array_buffer[15] := TO_BYTE(     TO_DWORD(buf4.Weld2Distance.UpperSuspect));

            array_buffer[16] := TO_BYTE(SHR(TO_DWORD(buf4.Weld2Distance.UpperBad), UINT#24));
            array_buffer[17] := TO_BYTE(SHR(TO_DWORD(buf4.Weld2Distance.UpperBad), UINT#16));
            array_buffer[18] := TO_BYTE(SHR(TO_DWORD(buf4.Weld2Distance.UpperBad),  UINT#8));
            array_buffer[19] := TO_BYTE(     TO_DWORD(buf4.Weld2Distance.UpperBad));

            // ---- Weld2Position.Enable bits → bytes 20..23 ----
            array_buffer[20].%X0 := buf4.Weld2Position.Enable._0;
            array_buffer[20].%X1 := buf4.Weld2Position.Enable._1;
            array_buffer[20].%X2 := buf4.Weld2Position.Enable._2;
            array_buffer[20].%X3 := buf4.Weld2Position.Enable._3;
            array_buffer[20].%X4 := buf4.Weld2Position.Enable._4;
            array_buffer[20].%X5 := buf4.Weld2Position.Enable._5;
            array_buffer[20].%X6 := buf4.Weld2Position.Enable._6;
            array_buffer[20].%X7 := buf4.Weld2Position.Enable._7;

            array_buffer[21].%X0 := buf4.Weld2Position.Enable._8;
            array_buffer[21].%X1 := buf4.Weld2Position.Enable._9;
            array_buffer[21].%X2 := buf4.Weld2Position.Enable._10;
            array_buffer[21].%X3 := buf4.Weld2Position.Enable._11;
            array_buffer[21].%X4 := buf4.Weld2Position.Enable._12;
            array_buffer[21].%X5 := buf4.Weld2Position.Enable._13;
            array_buffer[21].%X6 := buf4.Weld2Position.Enable._14;
            array_buffer[21].%X7 := buf4.Weld2Position.Enable._15;

            array_buffer[22].%X0 := buf4.Weld2Position.Enable._16;
            array_buffer[22].%X1 := buf4.Weld2Position.Enable._17;
            array_buffer[22].%X2 := buf4.Weld2Position.Enable._18;
            array_buffer[22].%X3 := buf4.Weld2Position.Enable._19;
            array_buffer[22].%X4 := buf4.Weld2Position.Enable._20;
            array_buffer[22].%X5 := buf4.Weld2Position.Enable._21;
            array_buffer[22].%X6 := buf4.Weld2Position.Enable._22;
            array_buffer[22].%X7 := buf4.Weld2Position.Enable._23;

            array_buffer[23].%X0 := buf4.Weld2Position.Enable.LowerBad_1;
            array_buffer[23].%X1 := buf4.Weld2Position.Enable.LowerSuspect_1;
            array_buffer[23].%X2 := buf4.Weld2Position.Enable.UpperSuspect_1;
            array_buffer[23].%X3 := buf4.Weld2Position.Enable.UpperBad_1;
            array_buffer[23].%X4 := buf4.Weld2Position.Enable.Display_1;
            array_buffer[23].%X5 := buf4.Weld2Position.Enable._29;
            array_buffer[23].%X6 := buf4.Weld2Position.Enable._30;
            array_buffer[23].%X7 := buf4.Weld2Position.Enable._31;

            // ---- Weld2Position (DINTs) → bytes 24..39 ----
            array_buffer[24] := TO_BYTE(SHR(TO_DWORD(buf4.Weld2Position.LowerBad), UINT#24));
            array_buffer[25] := TO_BYTE(SHR(TO_DWORD(buf4.Weld2Position.LowerBad), UINT#16));
            array_buffer[26] := TO_BYTE(SHR(TO_DWORD(buf4.Weld2Position.LowerBad),  UINT#8));
            array_buffer[27] := TO_BYTE(     TO_DWORD(buf4.Weld2Position.LowerBad));

            array_buffer[28] := TO_BYTE(SHR(TO_DWORD(buf4.Weld2Position.LowerSuspect), UINT#24));
            array_buffer[29] := TO_BYTE(SHR(TO_DWORD(buf4.Weld2Position.LowerSuspect), UINT#16));
            array_buffer[30] := TO_BYTE(SHR(TO_DWORD(buf4.Weld2Position.LowerSuspect),  UINT#8));
            array_buffer[31] := TO_BYTE(     TO_DWORD(buf4.Weld2Position.LowerSuspect));

            array_buffer[32] := TO_BYTE(SHR(TO_DWORD(buf4.Weld2Position.UpperSuspect), UINT#24));
            array_buffer[33] := TO_BYTE(SHR(TO_DWORD(buf4.Weld2Position.UpperSuspect), UINT#16));
            array_buffer[34] := TO_BYTE(SHR(TO_DWORD(buf4.Weld2Position.UpperSuspect),  UINT#8));
            array_buffer[35] := TO_BYTE(     TO_DWORD(buf4.Weld2Position.UpperSuspect));

            array_buffer[36] := TO_BYTE(SHR(TO_DWORD(buf4.Weld2Position.UpperBad), UINT#24));
            array_buffer[37] := TO_BYTE(SHR(TO_DWORD(buf4.Weld2Position.UpperBad), UINT#16));
            array_buffer[38] := TO_BYTE(SHR(TO_DWORD(buf4.Weld2Position.UpperBad),  UINT#8));
            array_buffer[39] := TO_BYTE(     TO_DWORD(buf4.Weld2Position.UpperBad));

            // ---- TotalWeldTime.Enable bits → bytes 40..43 ----
            array_buffer[40].%X0 := buf4.TotalWeldTime.Enable._0;
            array_buffer[40].%X1 := buf4.TotalWeldTime.Enable._1;
            array_buffer[40].%X2 := buf4.TotalWeldTime.Enable._2;
            array_buffer[40].%X3 := buf4.TotalWeldTime.Enable._3;
            array_buffer[40].%X4 := buf4.TotalWeldTime.Enable._4;
            array_buffer[40].%X5 := buf4.TotalWeldTime.Enable._5;
            array_buffer[40].%X6 := buf4.TotalWeldTime.Enable._6;
            array_buffer[40].%X7 := buf4.TotalWeldTime.Enable._7;

            array_buffer[41].%X0 := buf4.TotalWeldTime.Enable._8;
            array_buffer[41].%X1 := buf4.TotalWeldTime.Enable._9;
            array_buffer[41].%X2 := buf4.TotalWeldTime.Enable._10;
            array_buffer[41].%X3 := buf4.TotalWeldTime.Enable._11;
            array_buffer[41].%X4 := buf4.TotalWeldTime.Enable._12;
            array_buffer[41].%X5 := buf4.TotalWeldTime.Enable._13;
            array_buffer[41].%X6 := buf4.TotalWeldTime.Enable._14;
            array_buffer[41].%X7 := buf4.TotalWeldTime.Enable._15;

            array_buffer[42].%X0 := buf4.TotalWeldTime.Enable._16;
            array_buffer[42].%X1 := buf4.TotalWeldTime.Enable._17;
            array_buffer[42].%X2 := buf4.TotalWeldTime.Enable._18;
            array_buffer[42].%X3 := buf4.TotalWeldTime.Enable._19;
            array_buffer[42].%X4 := buf4.TotalWeldTime.Enable._20;
            array_buffer[42].%X5 := buf4.TotalWeldTime.Enable._21;
            array_buffer[42].%X6 := buf4.TotalWeldTime.Enable._22;
            array_buffer[42].%X7 := buf4.TotalWeldTime.Enable._23;

            array_buffer[43].%X0 := buf4.TotalWeldTime.Enable.LowerBad_1;
            array_buffer[43].%X1 := buf4.TotalWeldTime.Enable.LowerSuspect_1;
            array_buffer[43].%X2 := buf4.TotalWeldTime.Enable.UpperSuspect_1;
            array_buffer[43].%X3 := buf4.TotalWeldTime.Enable.UpperBad_1;
            array_buffer[43].%X4 := buf4.TotalWeldTime.Enable.Display_1;
            array_buffer[43].%X5 := buf4.TotalWeldTime.Enable._29;
            array_buffer[43].%X6 := buf4.TotalWeldTime.Enable._30;
            array_buffer[43].%X7 := buf4.TotalWeldTime.Enable._31;

            // ---- TotalWeldTime (DINTs) → bytes 44..59 ----
            array_buffer[44] := TO_BYTE(SHR(TO_DWORD(buf4.TotalWeldTime.LowerBad), UINT#24));
            array_buffer[45] := TO_BYTE(SHR(TO_DWORD(buf4.TotalWeldTime.LowerBad), UINT#16));
            array_buffer[46] := TO_BYTE(SHR(TO_DWORD(buf4.TotalWeldTime.LowerBad),  UINT#8));
            array_buffer[47] := TO_BYTE(     TO_DWORD(buf4.TotalWeldTime.LowerBad));

            array_buffer[48] := TO_BYTE(SHR(TO_DWORD(buf4.TotalWeldTime.LowerSuspect), UINT#24));
            array_buffer[49] := TO_BYTE(SHR(TO_DWORD(buf4.TotalWeldTime.LowerSuspect), UINT#16));
            array_buffer[50] := TO_BYTE(SHR(TO_DWORD(buf4.TotalWeldTime.LowerSuspect),  UINT#8));
            array_buffer[51] := TO_BYTE(     TO_DWORD(buf4.TotalWeldTime.LowerSuspect));

            array_buffer[52] := TO_BYTE(SHR(TO_DWORD(buf4.TotalWeldTime.UpperSuspect), UINT#24));
            array_buffer[53] := TO_BYTE(SHR(TO_DWORD(buf4.TotalWeldTime.UpperSuspect), UINT#16));
            array_buffer[54] := TO_BYTE(SHR(TO_DWORD(buf4.TotalWeldTime.UpperSuspect),  UINT#8));
            array_buffer[55] := TO_BYTE(     TO_DWORD(buf4.TotalWeldTime.UpperSuspect));

            array_buffer[56] := TO_BYTE(SHR(TO_DWORD(buf4.TotalWeldTime.UpperBad), UINT#24));
            array_buffer[57] := TO_BYTE(SHR(TO_DWORD(buf4.TotalWeldTime.UpperBad), UINT#16));
            array_buffer[58] := TO_BYTE(SHR(TO_DWORD(buf4.TotalWeldTime.UpperBad),  UINT#8));
            array_buffer[59] := TO_BYTE(     TO_DWORD(buf4.TotalWeldTime.UpperBad));

            // ---- TotalWeldEnergy.Enable bits → bytes 60..63 ----
            array_buffer[60].%X0 := buf4.TotalWeldEnergy.Enable._0;
            array_buffer[60].%X1 := buf4.TotalWeldEnergy.Enable._1;
            array_buffer[60].%X2 := buf4.TotalWeldEnergy.Enable._2;
            array_buffer[60].%X3 := buf4.TotalWeldEnergy.Enable._3;
            array_buffer[60].%X4 := buf4.TotalWeldEnergy.Enable._4;
            array_buffer[60].%X5 := buf4.TotalWeldEnergy.Enable._5;
            array_buffer[60].%X6 := buf4.TotalWeldEnergy.Enable._6;
            array_buffer[60].%X7 := buf4.TotalWeldEnergy.Enable._7;

            array_buffer[61].%X0 := buf4.TotalWeldEnergy.Enable._8;
            array_buffer[61].%X1 := buf4.TotalWeldEnergy.Enable._9;
            array_buffer[61].%X2 := buf4.TotalWeldEnergy.Enable._10;
            array_buffer[61].%X3 := buf4.TotalWeldEnergy.Enable._11;
            array_buffer[61].%X4 := buf4.TotalWeldEnergy.Enable._12;
            array_buffer[61].%X5 := buf4.TotalWeldEnergy.Enable._13;
            array_buffer[61].%X6 := buf4.TotalWeldEnergy.Enable._14;
            array_buffer[61].%X7 := buf4.TotalWeldEnergy.Enable._15;

            array_buffer[62].%X0 := buf4.TotalWeldEnergy.Enable._16;
            array_buffer[62].%X1 := buf4.TotalWeldEnergy.Enable._17;
            array_buffer[62].%X2 := buf4.TotalWeldEnergy.Enable._18;
            array_buffer[62].%X3 := buf4.TotalWeldEnergy.Enable._19;
            array_buffer[62].%X4 := buf4.TotalWeldEnergy.Enable._20;
            array_buffer[62].%X5 := buf4.TotalWeldEnergy.Enable._21;
            array_buffer[62].%X6 := buf4.TotalWeldEnergy.Enable._22;
            array_buffer[62].%X7 := buf4.TotalWeldEnergy.Enable._23;

            array_buffer[63].%X0 := buf4.TotalWeldEnergy.Enable.LowerBad_1;
            array_buffer[63].%X1 := buf4.TotalWeldEnergy.Enable.LowerSuspect_1;
            array_buffer[63].%X2 := buf4.TotalWeldEnergy.Enable.UpperSuspect_1;
            array_buffer[63].%X3 := buf4.TotalWeldEnergy.Enable.UpperBad_1;
            array_buffer[63].%X4 := buf4.TotalWeldEnergy.Enable.Display_1;
            array_buffer[63].%X5 := buf4.TotalWeldEnergy.Enable._29;
            array_buffer[63].%X6 := buf4.TotalWeldEnergy.Enable._30;
            array_buffer[63].%X7 := buf4.TotalWeldEnergy.Enable._31;

            // ---- TotalWeldEnergy (DINTs) → bytes 64..79 ----
            array_buffer[64] := TO_BYTE(SHR(TO_DWORD(buf4.TotalWeldEnergy.LowerBad), UINT#24));
            array_buffer[65] := TO_BYTE(SHR(TO_DWORD(buf4.TotalWeldEnergy.LowerBad), UINT#16));
            array_buffer[66] := TO_BYTE(SHR(TO_DWORD(buf4.TotalWeldEnergy.LowerBad),  UINT#8));
            array_buffer[67] := TO_BYTE(     TO_DWORD(buf4.TotalWeldEnergy.LowerBad));

            array_buffer[68] := TO_BYTE(SHR(TO_DWORD(buf4.TotalWeldEnergy.LowerSuspect), UINT#24));
            array_buffer[69] := TO_BYTE(SHR(TO_DWORD(buf4.TotalWeldEnergy.LowerSuspect), UINT#16));
            array_buffer[70] := TO_BYTE(SHR(TO_DWORD(buf4.TotalWeldEnergy.LowerSuspect),  UINT#8));
            array_buffer[71] := TO_BYTE(     TO_DWORD(buf4.TotalWeldEnergy.LowerSuspect));

            array_buffer[72] := TO_BYTE(SHR(TO_DWORD(buf4.TotalWeldEnergy.UpperSuspect), UINT#24));
            array_buffer[73] := TO_BYTE(SHR(TO_DWORD(buf4.TotalWeldEnergy.UpperSuspect), UINT#16));
            array_buffer[74] := TO_BYTE(SHR(TO_DWORD(buf4.TotalWeldEnergy.UpperSuspect),  UINT#8));
            array_buffer[75] := TO_BYTE(     TO_DWORD(buf4.TotalWeldEnergy.UpperSuspect));

            array_buffer[76] := TO_BYTE(SHR(TO_DWORD(buf4.TotalWeldEnergy.UpperBad), UINT#24));
            array_buffer[77] := TO_BYTE(SHR(TO_DWORD(buf4.TotalWeldEnergy.UpperBad), UINT#16));
            array_buffer[78] := TO_BYTE(SHR(TO_DWORD(buf4.TotalWeldEnergy.UpperBad),  UINT#8));
            array_buffer[79] := TO_BYTE(     TO_DWORD(buf4.TotalWeldEnergy.UpperBad));

            // ---- TotalWeldDistance.Enable bits → bytes 80..83 ----
            array_buffer[80].%X0 := buf4.TotalWeldDistance.Enable._0;
            array_buffer[80].%X1 := buf4.TotalWeldDistance.Enable._1;
            array_buffer[80].%X2 := buf4.TotalWeldDistance.Enable._2;
            array_buffer[80].%X3 := buf4.TotalWeldDistance.Enable._3;
            array_buffer[80].%X4 := buf4.TotalWeldDistance.Enable._4;
            array_buffer[80].%X5 := buf4.TotalWeldDistance.Enable._5;
            array_buffer[80].%X6 := buf4.TotalWeldDistance.Enable._6;
            array_buffer[80].%X7 := buf4.TotalWeldDistance.Enable._7;

            array_buffer[81].%X0 := buf4.TotalWeldDistance.Enable._8;
            array_buffer[81].%X1 := buf4.TotalWeldDistance.Enable._9;
            array_buffer[81].%X2 := buf4.TotalWeldDistance.Enable._10;
            array_buffer[81].%X3 := buf4.TotalWeldDistance.Enable._11;
            array_buffer[81].%X4 := buf4.TotalWeldDistance.Enable._12;
            array_buffer[81].%X5 := buf4.TotalWeldDistance.Enable._13;
            array_buffer[81].%X6 := buf4.TotalWeldDistance.Enable._14;
            array_buffer[81].%X7 := buf4.TotalWeldDistance.Enable._15;

            array_buffer[82].%X0 := buf4.TotalWeldDistance.Enable._16;
            array_buffer[82].%X1 := buf4.TotalWeldDistance.Enable._17;
            array_buffer[82].%X2 := buf4.TotalWeldDistance.Enable._18;
            array_buffer[82].%X3 := buf4.TotalWeldDistance.Enable._19;
            array_buffer[82].%X4 := buf4.TotalWeldDistance.Enable._20;
            array_buffer[82].%X5 := buf4.TotalWeldDistance.Enable._21;
            array_buffer[82].%X6 := buf4.TotalWeldDistance.Enable._22;
            array_buffer[82].%X7 := buf4.TotalWeldDistance.Enable._23;

            array_buffer[83].%X0 := buf4.TotalWeldDistance.Enable.LowerBad_1;
            array_buffer[83].%X1 := buf4.TotalWeldDistance.Enable.LowerSuspect_1;
            array_buffer[83].%X2 := buf4.TotalWeldDistance.Enable.UpperSuspect_1;
            array_buffer[83].%X3 := buf4.TotalWeldDistance.Enable.UpperBad_1;
            array_buffer[83].%X4 := buf4.TotalWeldDistance.Enable.Display_1;
            array_buffer[83].%X5 := buf4.TotalWeldDistance.Enable._29;
            array_buffer[83].%X6 := buf4.TotalWeldDistance.Enable._30;
            array_buffer[83].%X7 := buf4.TotalWeldDistance.Enable._31;

            // ---- TotalWeldDistance (DINTs) → bytes 84..99 ----
            array_buffer[84] := TO_BYTE(SHR(TO_DWORD(buf4.TotalWeldDistance.LowerBad), UINT#24));
            array_buffer[85] := TO_BYTE(SHR(TO_DWORD(buf4.TotalWeldDistance.LowerBad), UINT#16));
            array_buffer[86] := TO_BYTE(SHR(TO_DWORD(buf4.TotalWeldDistance.LowerBad),  UINT#8));
            array_buffer[87] := TO_BYTE(     TO_DWORD(buf4.TotalWeldDistance.LowerBad));

            array_buffer[88] := TO_BYTE(SHR(TO_DWORD(buf4.TotalWeldDistance.LowerSuspect), UINT#24));
            array_buffer[89] := TO_BYTE(SHR(TO_DWORD(buf4.TotalWeldDistance.LowerSuspect), UINT#16));
            array_buffer[90] := TO_BYTE(SHR(TO_DWORD(buf4.TotalWeldDistance.LowerSuspect),  UINT#8));
            array_buffer[91] := TO_BYTE(     TO_DWORD(buf4.TotalWeldDistance.LowerSuspect));

            array_buffer[92] := TO_BYTE(SHR(TO_DWORD(buf4.TotalWeldDistance.UpperSuspect), UINT#24));
            array_buffer[93] := TO_BYTE(SHR(TO_DWORD(buf4.TotalWeldDistance.UpperSuspect), UINT#16));
            array_buffer[94] := TO_BYTE(SHR(TO_DWORD(buf4.TotalWeldDistance.UpperSuspect),  UINT#8));
            array_buffer[95] := TO_BYTE(     TO_DWORD(buf4.TotalWeldDistance.UpperSuspect));

            array_buffer[96] := TO_BYTE(SHR(TO_DWORD(buf4.TotalWeldDistance.UpperBad), UINT#24));
            array_buffer[97] := TO_BYTE(SHR(TO_DWORD(buf4.TotalWeldDistance.UpperBad), UINT#16));
            array_buffer[98] := TO_BYTE(SHR(TO_DWORD(buf4.TotalWeldDistance.UpperBad),  UINT#8));
            array_buffer[99] := TO_BYTE(     TO_DWORD(buf4.TotalWeldDistance.UpperBad));

            // ---- DynamicHoldTime.Enable bits → bytes 100..103 ----
            array_buffer[100].%X0 := buf4.DynamicHoldTime.Enable._0;
            array_buffer[100].%X1 := buf4.DynamicHoldTime.Enable._1;
            array_buffer[100].%X2 := buf4.DynamicHoldTime.Enable._2;
            array_buffer[100].%X3 := buf4.DynamicHoldTime.Enable._3;
            array_buffer[100].%X4 := buf4.DynamicHoldTime.Enable._4;
            array_buffer[100].%X5 := buf4.DynamicHoldTime.Enable._5;
            array_buffer[100].%X6 := buf4.DynamicHoldTime.Enable._6;
            array_buffer[100].%X7 := buf4.DynamicHoldTime.Enable._7;

            array_buffer[101].%X0 := buf4.DynamicHoldTime.Enable._8;
            array_buffer[101].%X1 := buf4.DynamicHoldTime.Enable._9;
            array_buffer[101].%X2 := buf4.DynamicHoldTime.Enable._10;
            array_buffer[101].%X3 := buf4.DynamicHoldTime.Enable._11;
            array_buffer[101].%X4 := buf4.DynamicHoldTime.Enable._12;
            array_buffer[101].%X5 := buf4.DynamicHoldTime.Enable._13;
            array_buffer[101].%X6 := buf4.DynamicHoldTime.Enable._14;
            array_buffer[101].%X7 := buf4.DynamicHoldTime.Enable._15;

            array_buffer[102].%X0 := buf4.DynamicHoldTime.Enable._16;
            array_buffer[102].%X1 := buf4.DynamicHoldTime.Enable._17;
            array_buffer[102].%X2 := buf4.DynamicHoldTime.Enable._18;
            array_buffer[102].%X3 := buf4.DynamicHoldTime.Enable._19;
            array_buffer[102].%X4 := buf4.DynamicHoldTime.Enable._20;
            array_buffer[102].%X5 := buf4.DynamicHoldTime.Enable._21;
            array_buffer[102].%X6 := buf4.DynamicHoldTime.Enable._22;
            array_buffer[102].%X7 := buf4.DynamicHoldTime.Enable._23;

            array_buffer[103].%X0 := buf4.DynamicHoldTime.Enable.LowerBad_1;
            array_buffer[103].%X1 := buf4.DynamicHoldTime.Enable.LowerSuspect_1;
            array_buffer[103].%X2 := buf4.DynamicHoldTime.Enable.UpperSuspect_1;
            array_buffer[103].%X3 := buf4.DynamicHoldTime.Enable.UpperBad_1;
            array_buffer[103].%X4 := buf4.DynamicHoldTime.Enable.Display_1;
            array_buffer[103].%X5 := buf4.DynamicHoldTime.Enable._29;
            array_buffer[103].%X6 := buf4.DynamicHoldTime.Enable._30;
            array_buffer[103].%X7 := buf4.DynamicHoldTime.Enable._31;

            // ---- DynamicHoldTime (DINTs) → bytes 104..119 ----
            array_buffer[104] := TO_BYTE(SHR(TO_DWORD(buf4.DynamicHoldTime.LowerBad), UINT#24));
            array_buffer[105] := TO_BYTE(SHR(TO_DWORD(buf4.DynamicHoldTime.LowerBad), UINT#16));
            array_buffer[106] := TO_BYTE(SHR(TO_DWORD(buf4.DynamicHoldTime.LowerBad),  UINT#8));
            array_buffer[107] := TO_BYTE(     TO_DWORD(buf4.DynamicHoldTime.LowerBad));

            array_buffer[108] := TO_BYTE(SHR(TO_DWORD(buf4.DynamicHoldTime.LowerSuspect), UINT#24));
            array_buffer[109] := TO_BYTE(SHR(TO_DWORD(buf4.DynamicHoldTime.LowerSuspect), UINT#16));
            array_buffer[110] := TO_BYTE(SHR(TO_DWORD(buf4.DynamicHoldTime.LowerSuspect),  UINT#8));
            array_buffer[111] := TO_BYTE(     TO_DWORD(buf4.DynamicHoldTime.LowerSuspect));

            array_buffer[112] := TO_BYTE(SHR(TO_DWORD(buf4.DynamicHoldTime.UpperSuspect), UINT#24));
            array_buffer[113] := TO_BYTE(SHR(TO_DWORD(buf4.DynamicHoldTime.UpperSuspect), UINT#16));
            array_buffer[114] := TO_BYTE(SHR(TO_DWORD(buf4.DynamicHoldTime.UpperSuspect),  UINT#8));
            array_buffer[115] := TO_BYTE(     TO_DWORD(buf4.DynamicHoldTime.UpperSuspect));

            array_buffer[116] := TO_BYTE(SHR(TO_DWORD(buf4.DynamicHoldTime.UpperBad), UINT#24));
            array_buffer[117] := TO_BYTE(SHR(TO_DWORD(buf4.DynamicHoldTime.UpperBad), UINT#16));
            array_buffer[118] := TO_BYTE(SHR(TO_DWORD(buf4.DynamicHoldTime.UpperBad),  UINT#8));
            array_buffer[119] := TO_BYTE(     TO_DWORD(buf4.DynamicHoldTime.UpperBad));

            // ---- DynamicHoldDistance.Enable bits → bytes 120..123 ----
            array_buffer[120].%X0 := buf4.DynamicHoldDistance.Enable._0;
            array_buffer[120].%X1 := buf4.DynamicHoldDistance.Enable._1;
            array_buffer[120].%X2 := buf4.DynamicHoldDistance.Enable._2;
            array_buffer[120].%X3 := buf4.DynamicHoldDistance.Enable._3;
            array_buffer[120].%X4 := buf4.DynamicHoldDistance.Enable._4;
            array_buffer[120].%X5 := buf4.DynamicHoldDistance.Enable._5;
            array_buffer[120].%X6 := buf4.DynamicHoldDistance.Enable._6;
            array_buffer[120].%X7 := buf4.DynamicHoldDistance.Enable._7;

            array_buffer[121].%X0 := buf4.DynamicHoldDistance.Enable._8;
            array_buffer[121].%X1 := buf4.DynamicHoldDistance.Enable._9;
            array_buffer[121].%X2 := buf4.DynamicHoldDistance.Enable._10;
            array_buffer[121].%X3 := buf4.DynamicHoldDistance.Enable._11;
            array_buffer[121].%X4 := buf4.DynamicHoldDistance.Enable._12;
            array_buffer[121].%X5 := buf4.DynamicHoldDistance.Enable._13;
            array_buffer[121].%X6 := buf4.DynamicHoldDistance.Enable._14;
            array_buffer[121].%X7 := buf4.DynamicHoldDistance.Enable._15;

            array_buffer[122].%X0 := buf4.DynamicHoldDistance.Enable._16;
            array_buffer[122].%X1 := buf4.DynamicHoldDistance.Enable._17;
            array_buffer[122].%X2 := buf4.DynamicHoldDistance.Enable._18;
            array_buffer[122].%X3 := buf4.DynamicHoldDistance.Enable._19;
            array_buffer[122].%X4 := buf4.DynamicHoldDistance.Enable._20;
            array_buffer[122].%X5 := buf4.DynamicHoldDistance.Enable._21;
            array_buffer[122].%X6 := buf4.DynamicHoldDistance.Enable._22;
            array_buffer[122].%X7 := buf4.DynamicHoldDistance.Enable._23;

            array_buffer[123].%X0 := buf4.DynamicHoldDistance.Enable.LowerBad_1;
            array_buffer[123].%X1 := buf4.DynamicHoldDistance.Enable.LowerSuspect_1;
            array_buffer[123].%X2 := buf4.DynamicHoldDistance.Enable.UpperSuspect_1;
            array_buffer[123].%X3 := buf4.DynamicHoldDistance.Enable.UpperBad_1;
            array_buffer[123].%X4 := buf4.DynamicHoldDistance.Enable.Display_1;
            array_buffer[123].%X5 := buf4.DynamicHoldDistance.Enable._29;
            array_buffer[123].%X6 := buf4.DynamicHoldDistance.Enable._30;
            array_buffer[123].%X7 := buf4.DynamicHoldDistance.Enable._31;

            // ---- DynamicHoldDistance (DINTs) → bytes 124..139 ----
            array_buffer[124] := TO_BYTE(SHR(TO_DWORD(buf4.DynamicHoldDistance.LowerBad), UINT#24));
            array_buffer[125] := TO_BYTE(SHR(TO_DWORD(buf4.DynamicHoldDistance.LowerBad), UINT#16));
            array_buffer[126] := TO_BYTE(SHR(TO_DWORD(buf4.DynamicHoldDistance.LowerBad),  UINT#8));
            array_buffer[127] := TO_BYTE(     TO_DWORD(buf4.DynamicHoldDistance.LowerBad));

            array_buffer[128] := TO_BYTE(SHR(TO_DWORD(buf4.DynamicHoldDistance.LowerSuspect), UINT#24));
            array_buffer[129] := TO_BYTE(SHR(TO_DWORD(buf4.DynamicHoldDistance.LowerSuspect), UINT#16));
            array_buffer[130] := TO_BYTE(SHR(TO_DWORD(buf4.DynamicHoldDistance.LowerSuspect),  UINT#8));
            array_buffer[131] := TO_BYTE(     TO_DWORD(buf4.DynamicHoldDistance.LowerSuspect));

            array_buffer[132] := TO_BYTE(SHR(TO_DWORD(buf4.DynamicHoldDistance.UpperSuspect), UINT#24));
            array_buffer[133] := TO_BYTE(SHR(TO_DWORD(buf4.DynamicHoldDistance.UpperSuspect), UINT#16));
            array_buffer[134] := TO_BYTE(SHR(TO_DWORD(buf4.DynamicHoldDistance.UpperSuspect),  UINT#8));
            array_buffer[135] := TO_BYTE(     TO_DWORD(buf4.DynamicHoldDistance.UpperSuspect));

            array_buffer[136] := TO_BYTE(SHR(TO_DWORD(buf4.DynamicHoldDistance.UpperBad), UINT#24));
            array_buffer[137] := TO_BYTE(SHR(TO_DWORD(buf4.DynamicHoldDistance.UpperBad), UINT#16));
            array_buffer[138] := TO_BYTE(SHR(TO_DWORD(buf4.DynamicHoldDistance.UpperBad),  UINT#8));
            array_buffer[139] := TO_BYTE(     TO_DWORD(buf4.DynamicHoldDistance.UpperBad));

            // ---- TotalCycleTime.Enable bits → bytes 140..143 ----
            array_buffer[140].%X0 := buf4.TotalCycleTime.Enable._0;
            array_buffer[140].%X1 := buf4.TotalCycleTime.Enable._1;
            array_buffer[140].%X2 := buf4.TotalCycleTime.Enable._2;
            array_buffer[140].%X3 := buf4.TotalCycleTime.Enable._3;
            array_buffer[140].%X4 := buf4.TotalCycleTime.Enable._4;
            array_buffer[140].%X5 := buf4.TotalCycleTime.Enable._5;
            array_buffer[140].%X6 := buf4.TotalCycleTime.Enable._6;
            array_buffer[140].%X7 := buf4.TotalCycleTime.Enable._7;

            array_buffer[141].%X0 := buf4.TotalCycleTime.Enable._8;
            array_buffer[141].%X1 := buf4.TotalCycleTime.Enable._9;
            array_buffer[141].%X2 := buf4.TotalCycleTime.Enable._10;
            array_buffer[141].%X3 := buf4.TotalCycleTime.Enable._11;
            array_buffer[141].%X4 := buf4.TotalCycleTime.Enable._12;
            array_buffer[141].%X5 := buf4.TotalCycleTime.Enable._13;
            array_buffer[141].%X6 := buf4.TotalCycleTime.Enable._14;
            array_buffer[141].%X7 := buf4.TotalCycleTime.Enable._15;

            array_buffer[142].%X0 := buf4.TotalCycleTime.Enable._16;
            array_buffer[142].%X1 := buf4.TotalCycleTime.Enable._17;
            array_buffer[142].%X2 := buf4.TotalCycleTime.Enable._18;
            array_buffer[142].%X3 := buf4.TotalCycleTime.Enable._19;
            array_buffer[142].%X4 := buf4.TotalCycleTime.Enable._20;
            array_buffer[142].%X5 := buf4.TotalCycleTime.Enable._21;
            array_buffer[142].%X6 := buf4.TotalCycleTime.Enable._22;
            array_buffer[142].%X7 := buf4.TotalCycleTime.Enable._23;

            array_buffer[143].%X0 := buf4.TotalCycleTime.Enable.LowerBad_1;
            array_buffer[143].%X1 := buf4.TotalCycleTime.Enable.LowerSuspect_1;
            array_buffer[143].%X2 := buf4.TotalCycleTime.Enable.UpperSuspect_1;
            array_buffer[143].%X3 := buf4.TotalCycleTime.Enable.UpperBad_1;
            array_buffer[143].%X4 := buf4.TotalCycleTime.Enable.Display_1;
            array_buffer[143].%X5 := buf4.TotalCycleTime.Enable._29;
            array_buffer[143].%X6 := buf4.TotalCycleTime.Enable._30;
            array_buffer[143].%X7 := buf4.TotalCycleTime.Enable._31;

            // ---- TotalCycleTime (DINTs) → bytes 144..159 ----
            array_buffer[144] := TO_BYTE(SHR(TO_DWORD(buf4.TotalCycleTime.LowerBad), UINT#24));
            array_buffer[145] := TO_BYTE(SHR(TO_DWORD(buf4.TotalCycleTime.LowerBad), UINT#16));
            array_buffer[146] := TO_BYTE(SHR(TO_DWORD(buf4.TotalCycleTime.LowerBad),  UINT#8));
            array_buffer[147] := TO_BYTE(     TO_DWORD(buf4.TotalCycleTime.LowerBad));

            array_buffer[148] := TO_BYTE(SHR(TO_DWORD(buf4.TotalCycleTime.LowerSuspect), UINT#24));
            array_buffer[149] := TO_BYTE(SHR(TO_DWORD(buf4.TotalCycleTime.LowerSuspect), UINT#16));
            array_buffer[150] := TO_BYTE(SHR(TO_DWORD(buf4.TotalCycleTime.LowerSuspect),  UINT#8));
            array_buffer[151] := TO_BYTE(     TO_DWORD(buf4.TotalCycleTime.LowerSuspect));

            array_buffer[152] := TO_BYTE(SHR(TO_DWORD(buf4.TotalCycleTime.UpperSuspect), UINT#24));
            array_buffer[153] := TO_BYTE(SHR(TO_DWORD(buf4.TotalCycleTime.UpperSuspect), UINT#16));
            array_buffer[154] := TO_BYTE(SHR(TO_DWORD(buf4.TotalCycleTime.UpperSuspect),  UINT#8));
            array_buffer[155] := TO_BYTE(     TO_DWORD(buf4.TotalCycleTime.UpperSuspect));

            array_buffer[156] := TO_BYTE(SHR(TO_DWORD(buf4.TotalCycleTime.UpperBad), UINT#24));
            array_buffer[157] := TO_BYTE(SHR(TO_DWORD(buf4.TotalCycleTime.UpperBad), UINT#16));
            array_buffer[158] := TO_BYTE(SHR(TO_DWORD(buf4.TotalCycleTime.UpperBad),  UINT#8));
            array_buffer[159] := TO_BYTE(     TO_DWORD(buf4.TotalCycleTime.UpperBad));

            // ---- FinalHoldPosition.Enable bits → bytes 160..163 ----
            array_buffer[160].%X0 := buf4.FinalHoldPosition.Enable._0;
            array_buffer[160].%X1 := buf4.FinalHoldPosition.Enable._1;
            array_buffer[160].%X2 := buf4.FinalHoldPosition.Enable._2;
            array_buffer[160].%X3 := buf4.FinalHoldPosition.Enable._3;
            array_buffer[160].%X4 := buf4.FinalHoldPosition.Enable._4;
            array_buffer[160].%X5 := buf4.FinalHoldPosition.Enable._5;
            array_buffer[160].%X6 := buf4.FinalHoldPosition.Enable._6;
            array_buffer[160].%X7 := buf4.FinalHoldPosition.Enable._7;

            array_buffer[161].%X0 := buf4.FinalHoldPosition.Enable._8;
            array_buffer[161].%X1 := buf4.FinalHoldPosition.Enable._9;
            array_buffer[161].%X2 := buf4.FinalHoldPosition.Enable._10;
            array_buffer[161].%X3 := buf4.FinalHoldPosition.Enable._11;
            array_buffer[161].%X4 := buf4.FinalHoldPosition.Enable._12;
            array_buffer[161].%X5 := buf4.FinalHoldPosition.Enable._13;
            array_buffer[161].%X6 := buf4.FinalHoldPosition.Enable._14;
            array_buffer[161].%X7 := buf4.FinalHoldPosition.Enable._15;

            array_buffer[162].%X0 := buf4.FinalHoldPosition.Enable._16;
            array_buffer[162].%X1 := buf4.FinalHoldPosition.Enable._17;
            array_buffer[162].%X2 := buf4.FinalHoldPosition.Enable._18;
            array_buffer[162].%X3 := buf4.FinalHoldPosition.Enable._19;
            array_buffer[162].%X4 := buf4.FinalHoldPosition.Enable._20;
            array_buffer[162].%X5 := buf4.FinalHoldPosition.Enable._21;
            array_buffer[162].%X6 := buf4.FinalHoldPosition.Enable._22;
            array_buffer[162].%X7 := buf4.FinalHoldPosition.Enable._23;

            array_buffer[163].%X0 := buf4.FinalHoldPosition.Enable.LowerBad_1;
            array_buffer[163].%X1 := buf4.FinalHoldPosition.Enable.LowerSuspect_1;
            array_buffer[163].%X2 := buf4.FinalHoldPosition.Enable.UpperSuspect_1;
            array_buffer[163].%X3 := buf4.FinalHoldPosition.Enable.UpperBad_1;
            array_buffer[163].%X4 := buf4.FinalHoldPosition.Enable.Display_1;
            array_buffer[163].%X5 := buf4.FinalHoldPosition.Enable._29;
            array_buffer[163].%X6 := buf4.FinalHoldPosition.Enable._30;
            array_buffer[163].%X7 := buf4.FinalHoldPosition.Enable._31;

            // ---- FinalHoldPosition (DINTs) → bytes 164..179 ----
            array_buffer[164] := TO_BYTE(SHR(TO_DWORD(buf4.FinalHoldPosition.LowerBad), UINT#24));
            array_buffer[165] := TO_BYTE(SHR(TO_DWORD(buf4.FinalHoldPosition.LowerBad), UINT#16));
            array_buffer[166] := TO_BYTE(SHR(TO_DWORD(buf4.FinalHoldPosition.LowerBad),  UINT#8));
            array_buffer[167] := TO_BYTE(     TO_DWORD(buf4.FinalHoldPosition.LowerBad));

            array_buffer[168] := TO_BYTE(SHR(TO_DWORD(buf4.FinalHoldPosition.LowerSuspect), UINT#24));
            array_buffer[169] := TO_BYTE(SHR(TO_DWORD(buf4.FinalHoldPosition.LowerSuspect), UINT#16));
            array_buffer[170] := TO_BYTE(SHR(TO_DWORD(buf4.FinalHoldPosition.LowerSuspect),  UINT#8));
            array_buffer[171] := TO_BYTE(     TO_DWORD(buf4.FinalHoldPosition.LowerSuspect));

            array_buffer[172] := TO_BYTE(SHR(TO_DWORD(buf4.FinalHoldPosition.UpperSuspect), UINT#24));
            array_buffer[173] := TO_BYTE(SHR(TO_DWORD(buf4.FinalHoldPosition.UpperSuspect), UINT#16));
            array_buffer[174] := TO_BYTE(SHR(TO_DWORD(buf4.FinalHoldPosition.UpperSuspect),  UINT#8));
            array_buffer[175] := TO_BYTE(     TO_DWORD(buf4.FinalHoldPosition.UpperSuspect));

            array_buffer[176] := TO_BYTE(SHR(TO_DWORD(buf4.FinalHoldPosition.UpperBad), UINT#24));
            array_buffer[177] := TO_BYTE(SHR(TO_DWORD(buf4.FinalHoldPosition.UpperBad), UINT#16));
            array_buffer[178] := TO_BYTE(SHR(TO_DWORD(buf4.FinalHoldPosition.UpperBad),  UINT#8));
            array_buffer[179] := TO_BYTE(     TO_DWORD(buf4.FinalHoldPosition.UpperBad));

            // ---- ErrorStatus.Enable bits → bytes 180..183 ----
            array_buffer[180].%X0 := buf4.ErrorStatus.Enable._0;
            array_buffer[180].%X1 := buf4.ErrorStatus.Enable._1;
            array_buffer[180].%X2 := buf4.ErrorStatus.Enable._2;
            array_buffer[180].%X3 := buf4.ErrorStatus.Enable._3;
            array_buffer[180].%X4 := buf4.ErrorStatus.Enable._4;
            array_buffer[180].%X5 := buf4.ErrorStatus.Enable._5;
            array_buffer[180].%X6 := buf4.ErrorStatus.Enable._6;
            array_buffer[180].%X7 := buf4.ErrorStatus.Enable._7;

            array_buffer[181].%X0 := buf4.ErrorStatus.Enable._8;
            array_buffer[181].%X1 := buf4.ErrorStatus.Enable._9;
            array_buffer[181].%X2 := buf4.ErrorStatus.Enable._10;
            array_buffer[181].%X3 := buf4.ErrorStatus.Enable._11;
            array_buffer[181].%X4 := buf4.ErrorStatus.Enable._12;
            array_buffer[181].%X5 := buf4.ErrorStatus.Enable._13;
            array_buffer[181].%X6 := buf4.ErrorStatus.Enable._14;
            array_buffer[181].%X7 := buf4.ErrorStatus.Enable._15;

            array_buffer[182].%X0 := buf4.ErrorStatus.Enable._16;
            array_buffer[182].%X1 := buf4.ErrorStatus.Enable._17;
            array_buffer[182].%X2 := buf4.ErrorStatus.Enable._18;
            array_buffer[182].%X3 := buf4.ErrorStatus.Enable._19;
            array_buffer[182].%X4 := buf4.ErrorStatus.Enable._20;
            array_buffer[182].%X5 := buf4.ErrorStatus.Enable._21;
            array_buffer[182].%X6 := buf4.ErrorStatus.Enable._22;
            array_buffer[182].%X7 := buf4.ErrorStatus.Enable._23;

            array_buffer[183].%X0 := buf4.ErrorStatus.Enable.LowerBad_1;
            array_buffer[183].%X1 := buf4.ErrorStatus.Enable.LowerSuspect_1;
            array_buffer[183].%X2 := buf4.ErrorStatus.Enable.UpperSuspect_1;
            array_buffer[183].%X3 := buf4.ErrorStatus.Enable.UpperBad_1;
            array_buffer[183].%X4 := buf4.ErrorStatus.Enable.Display_1;
            array_buffer[183].%X5 := buf4.ErrorStatus.Enable._29;
            array_buffer[183].%X6 := buf4.ErrorStatus.Enable._30;
            array_buffer[183].%X7 := buf4.ErrorStatus.Enable._31;

            // ---- ErrorStatus (DINTs) → bytes 184..199 ----
            array_buffer[184] := TO_BYTE(SHR(TO_DWORD(buf4.ErrorStatus.LowerBad), UINT#24));
            array_buffer[185] := TO_BYTE(SHR(TO_DWORD(buf4.ErrorStatus.LowerBad), UINT#16));
            array_buffer[186] := TO_BYTE(SHR(TO_DWORD(buf4.ErrorStatus.LowerBad),  UINT#8));
            array_buffer[187] := TO_BYTE(     TO_DWORD(buf4.ErrorStatus.LowerBad));

            array_buffer[188] := TO_BYTE(SHR(TO_DWORD(buf4.ErrorStatus.LowerSuspect), UINT#24));
            array_buffer[189] := TO_BYTE(SHR(TO_DWORD(buf4.ErrorStatus.LowerSuspect), UINT#16));
            array_buffer[190] := TO_BYTE(SHR(TO_DWORD(buf4.ErrorStatus.LowerSuspect),  UINT#8));
            array_buffer[191] := TO_BYTE(     TO_DWORD(buf4.ErrorStatus.LowerSuspect));

            array_buffer[192] := TO_BYTE(SHR(TO_DWORD(buf4.ErrorStatus.UpperSuspect), UINT#24));
            array_buffer[193] := TO_BYTE(SHR(TO_DWORD(buf4.ErrorStatus.UpperSuspect), UINT#16));
            array_buffer[194] := TO_BYTE(SHR(TO_DWORD(buf4.ErrorStatus.UpperSuspect),  UINT#8));
            array_buffer[195] := TO_BYTE(     TO_DWORD(buf4.ErrorStatus.UpperSuspect));

            array_buffer[196] := TO_BYTE(SHR(TO_DWORD(buf4.ErrorStatus.UpperBad), UINT#24));
            array_buffer[197] := TO_BYTE(SHR(TO_DWORD(buf4.ErrorStatus.UpperBad), UINT#16));
            array_buffer[198] := TO_BYTE(SHR(TO_DWORD(buf4.ErrorStatus.UpperBad),  UINT#8));
            array_buffer[199] := TO_BYTE(     TO_DWORD(buf4.ErrorStatus.UpperBad));

        END_METHOD

        METHOD PRIVATE buf5_TO_ByteArray
            VAR_IN_OUT
                buf5 : Axo_IQ_SeriesWelder_data5_176bytes;
                array_buffer : ARRAY[0..253] OF BYTE;
            END_VAR

            // --- Sensor[1] (bytes 0..19) ---
            array_buffer[ 0] := TO_BYTE(SHR(TO_DWORD(buf5.AnalogSensor.Sensor[1].Enable),    UINT#24));
            array_buffer[ 1] := TO_BYTE(SHR(TO_DWORD(buf5.AnalogSensor.Sensor[1].Enable),    UINT#16));
            array_buffer[ 2] := TO_BYTE(SHR(TO_DWORD(buf5.AnalogSensor.Sensor[1].Enable),     UINT#8));
            array_buffer[ 3] := TO_BYTE(     TO_DWORD(buf5.AnalogSensor.Sensor[1].Enable));

            array_buffer[ 4] := TO_BYTE(SHR(TO_DWORD(buf5.AnalogSensor.Sensor[1].MIN_VOLT),  UINT#24));
            array_buffer[ 5] := TO_BYTE(SHR(TO_DWORD(buf5.AnalogSensor.Sensor[1].MIN_VOLT),  UINT#16));
            array_buffer[ 6] := TO_BYTE(SHR(TO_DWORD(buf5.AnalogSensor.Sensor[1].MIN_VOLT),   UINT#8));
            array_buffer[ 7] := TO_BYTE(     TO_DWORD(buf5.AnalogSensor.Sensor[1].MIN_VOLT));

            array_buffer[ 8] := TO_BYTE(SHR(TO_DWORD(buf5.AnalogSensor.Sensor[1].MAX_VOLT),  UINT#24));
            array_buffer[ 9] := TO_BYTE(SHR(TO_DWORD(buf5.AnalogSensor.Sensor[1].MAX_VOLT),  UINT#16));
            array_buffer[10] := TO_BYTE(SHR(TO_DWORD(buf5.AnalogSensor.Sensor[1].MAX_VOLT),   UINT#8));
            array_buffer[11] := TO_BYTE(     TO_DWORD(buf5.AnalogSensor.Sensor[1].MAX_VOLT));

            array_buffer[12] := TO_BYTE(SHR(TO_DWORD(buf5.AnalogSensor.Sensor[1].MIN_VAL),   UINT#24));
            array_buffer[13] := TO_BYTE(SHR(TO_DWORD(buf5.AnalogSensor.Sensor[1].MIN_VAL),   UINT#16));
            array_buffer[14] := TO_BYTE(SHR(TO_DWORD(buf5.AnalogSensor.Sensor[1].MIN_VAL),    UINT#8));
            array_buffer[15] := TO_BYTE(     TO_DWORD(buf5.AnalogSensor.Sensor[1].MIN_VAL));

            array_buffer[16] := TO_BYTE(SHR(TO_DWORD(buf5.AnalogSensor.Sensor[1].MAX_VAL),   UINT#24));
            array_buffer[17] := TO_BYTE(SHR(TO_DWORD(buf5.AnalogSensor.Sensor[1].MAX_VAL),   UINT#16));
            array_buffer[18] := TO_BYTE(SHR(TO_DWORD(buf5.AnalogSensor.Sensor[1].MAX_VAL),    UINT#8));
            array_buffer[19] := TO_BYTE(     TO_DWORD(buf5.AnalogSensor.Sensor[1].MAX_VAL));

            // --- Sensor[2] (bytes 20..39) ---
            array_buffer[20] := TO_BYTE(SHR(TO_DWORD(buf5.AnalogSensor.Sensor[2].Enable),    UINT#24));
            array_buffer[21] := TO_BYTE(SHR(TO_DWORD(buf5.AnalogSensor.Sensor[2].Enable),    UINT#16));
            array_buffer[22] := TO_BYTE(SHR(TO_DWORD(buf5.AnalogSensor.Sensor[2].Enable),     UINT#8));
            array_buffer[23] := TO_BYTE(     TO_DWORD(buf5.AnalogSensor.Sensor[2].Enable));

            array_buffer[24] := TO_BYTE(SHR(TO_DWORD(buf5.AnalogSensor.Sensor[2].MIN_VOLT),  UINT#24));
            array_buffer[25] := TO_BYTE(SHR(TO_DWORD(buf5.AnalogSensor.Sensor[2].MIN_VOLT),  UINT#16));
            array_buffer[26] := TO_BYTE(SHR(TO_DWORD(buf5.AnalogSensor.Sensor[2].MIN_VOLT),   UINT#8));
            array_buffer[27] := TO_BYTE(     TO_DWORD(buf5.AnalogSensor.Sensor[2].MIN_VOLT));

            array_buffer[28] := TO_BYTE(SHR(TO_DWORD(buf5.AnalogSensor.Sensor[2].MAX_VOLT),  UINT#24));
            array_buffer[29] := TO_BYTE(SHR(TO_DWORD(buf5.AnalogSensor.Sensor[2].MAX_VOLT),  UINT#16));
            array_buffer[30] := TO_BYTE(SHR(TO_DWORD(buf5.AnalogSensor.Sensor[2].MAX_VOLT),   UINT#8));
            array_buffer[31] := TO_BYTE(     TO_DWORD(buf5.AnalogSensor.Sensor[2].MAX_VOLT));

            array_buffer[32] := TO_BYTE(SHR(TO_DWORD(buf5.AnalogSensor.Sensor[2].MIN_VAL),   UINT#24));
            array_buffer[33] := TO_BYTE(SHR(TO_DWORD(buf5.AnalogSensor.Sensor[2].MIN_VAL),   UINT#16));
            array_buffer[34] := TO_BYTE(SHR(TO_DWORD(buf5.AnalogSensor.Sensor[2].MIN_VAL),    UINT#8));
            array_buffer[35] := TO_BYTE(     TO_DWORD(buf5.AnalogSensor.Sensor[2].MIN_VAL));

            array_buffer[36] := TO_BYTE(SHR(TO_DWORD(buf5.AnalogSensor.Sensor[2].MAX_VAL),   UINT#24));
            array_buffer[37] := TO_BYTE(SHR(TO_DWORD(buf5.AnalogSensor.Sensor[2].MAX_VAL),   UINT#16));
            array_buffer[38] := TO_BYTE(SHR(TO_DWORD(buf5.AnalogSensor.Sensor[2].MAX_VAL),    UINT#8));
            array_buffer[39] := TO_BYTE(     TO_DWORD(buf5.AnalogSensor.Sensor[2].MAX_VAL));

            // --- Sensor[3] (bytes 40..59) ---
            array_buffer[40] := TO_BYTE(SHR(TO_DWORD(buf5.AnalogSensor.Sensor[3].Enable),    UINT#24));
            array_buffer[41] := TO_BYTE(SHR(TO_DWORD(buf5.AnalogSensor.Sensor[3].Enable),    UINT#16));
            array_buffer[42] := TO_BYTE(SHR(TO_DWORD(buf5.AnalogSensor.Sensor[3].Enable),     UINT#8));
            array_buffer[43] := TO_BYTE(     TO_DWORD(buf5.AnalogSensor.Sensor[3].Enable));

            array_buffer[44] := TO_BYTE(SHR(TO_DWORD(buf5.AnalogSensor.Sensor[3].MIN_VOLT),  UINT#24));
            array_buffer[45] := TO_BYTE(SHR(TO_DWORD(buf5.AnalogSensor.Sensor[3].MIN_VOLT),  UINT#16));
            array_buffer[46] := TO_BYTE(SHR(TO_DWORD(buf5.AnalogSensor.Sensor[3].MIN_VOLT),   UINT#8));
            array_buffer[47] := TO_BYTE(     TO_DWORD(buf5.AnalogSensor.Sensor[3].MIN_VOLT));

            array_buffer[48] := TO_BYTE(SHR(TO_DWORD(buf5.AnalogSensor.Sensor[3].MAX_VOLT),  UINT#24));
            array_buffer[49] := TO_BYTE(SHR(TO_DWORD(buf5.AnalogSensor.Sensor[3].MAX_VOLT),  UINT#16));
            array_buffer[50] := TO_BYTE(SHR(TO_DWORD(buf5.AnalogSensor.Sensor[3].MAX_VOLT),   UINT#8));
            array_buffer[51] := TO_BYTE(     TO_DWORD(buf5.AnalogSensor.Sensor[3].MAX_VOLT));

            array_buffer[52] := TO_BYTE(SHR(TO_DWORD(buf5.AnalogSensor.Sensor[3].MIN_VAL),   UINT#24));
            array_buffer[53] := TO_BYTE(SHR(TO_DWORD(buf5.AnalogSensor.Sensor[3].MIN_VAL),   UINT#16));
            array_buffer[54] := TO_BYTE(SHR(TO_DWORD(buf5.AnalogSensor.Sensor[3].MIN_VAL),    UINT#8));
            array_buffer[55] := TO_BYTE(     TO_DWORD(buf5.AnalogSensor.Sensor[3].MIN_VAL));

            array_buffer[56] := TO_BYTE(SHR(TO_DWORD(buf5.AnalogSensor.Sensor[3].MAX_VAL),   UINT#24));
            array_buffer[57] := TO_BYTE(SHR(TO_DWORD(buf5.AnalogSensor.Sensor[3].MAX_VAL),   UINT#16));
            array_buffer[58] := TO_BYTE(SHR(TO_DWORD(buf5.AnalogSensor.Sensor[3].MAX_VAL),    UINT#8));
            array_buffer[59] := TO_BYTE(     TO_DWORD(buf5.AnalogSensor.Sensor[3].MAX_VAL));

            // --- Sensor[4] (bytes 60..79) ---
            array_buffer[60] := TO_BYTE(SHR(TO_DWORD(buf5.AnalogSensor.Sensor[4].Enable),    UINT#24));
            array_buffer[61] := TO_BYTE(SHR(TO_DWORD(buf5.AnalogSensor.Sensor[4].Enable),    UINT#16));
            array_buffer[62] := TO_BYTE(SHR(TO_DWORD(buf5.AnalogSensor.Sensor[4].Enable),     UINT#8));
            array_buffer[63] := TO_BYTE(     TO_DWORD(buf5.AnalogSensor.Sensor[4].Enable));

            array_buffer[64] := TO_BYTE(SHR(TO_DWORD(buf5.AnalogSensor.Sensor[4].MIN_VOLT),  UINT#24));
            array_buffer[65] := TO_BYTE(SHR(TO_DWORD(buf5.AnalogSensor.Sensor[4].MIN_VOLT),  UINT#16));
            array_buffer[66] := TO_BYTE(SHR(TO_DWORD(buf5.AnalogSensor.Sensor[4].MIN_VOLT),   UINT#8));
            array_buffer[67] := TO_BYTE(     TO_DWORD(buf5.AnalogSensor.Sensor[4].MIN_VOLT));

            array_buffer[68] := TO_BYTE(SHR(TO_DWORD(buf5.AnalogSensor.Sensor[4].MAX_VOLT),  UINT#24));
            array_buffer[69] := TO_BYTE(SHR(TO_DWORD(buf5.AnalogSensor.Sensor[4].MAX_VOLT),  UINT#16));
            array_buffer[70] := TO_BYTE(SHR(TO_DWORD(buf5.AnalogSensor.Sensor[4].MAX_VOLT),   UINT#8));
            array_buffer[71] := TO_BYTE(     TO_DWORD(buf5.AnalogSensor.Sensor[4].MAX_VOLT));

            array_buffer[72] := TO_BYTE(SHR(TO_DWORD(buf5.AnalogSensor.Sensor[4].MIN_VAL),   UINT#24));
            array_buffer[73] := TO_BYTE(SHR(TO_DWORD(buf5.AnalogSensor.Sensor[4].MIN_VAL),   UINT#16));
            array_buffer[74] := TO_BYTE(SHR(TO_DWORD(buf5.AnalogSensor.Sensor[4].MIN_VAL),    UINT#8));
            array_buffer[75] := TO_BYTE(     TO_DWORD(buf5.AnalogSensor.Sensor[4].MIN_VAL));

            array_buffer[76] := TO_BYTE(SHR(TO_DWORD(buf5.AnalogSensor.Sensor[4].MAX_VAL),   UINT#24));
            array_buffer[77] := TO_BYTE(SHR(TO_DWORD(buf5.AnalogSensor.Sensor[4].MAX_VAL),   UINT#16));
            array_buffer[78] := TO_BYTE(SHR(TO_DWORD(buf5.AnalogSensor.Sensor[4].MAX_VAL),    UINT#8));
            array_buffer[79] := TO_BYTE(     TO_DWORD(buf5.AnalogSensor.Sensor[4].MAX_VAL));

            // --- Sensor[5] (bytes 80..99) ---
            array_buffer[80] := TO_BYTE(SHR(TO_DWORD(buf5.AnalogSensor.Sensor[5].Enable),    UINT#24));
            array_buffer[81] := TO_BYTE(SHR(TO_DWORD(buf5.AnalogSensor.Sensor[5].Enable),    UINT#16));
            array_buffer[82] := TO_BYTE(SHR(TO_DWORD(buf5.AnalogSensor.Sensor[5].Enable),     UINT#8));
            array_buffer[83] := TO_BYTE(     TO_DWORD(buf5.AnalogSensor.Sensor[5].Enable));

            array_buffer[84] := TO_BYTE(SHR(TO_DWORD(buf5.AnalogSensor.Sensor[5].MIN_VOLT),  UINT#24));
            array_buffer[85] := TO_BYTE(SHR(TO_DWORD(buf5.AnalogSensor.Sensor[5].MIN_VOLT),  UINT#16));
            array_buffer[86] := TO_BYTE(SHR(TO_DWORD(buf5.AnalogSensor.Sensor[5].MIN_VOLT),   UINT#8));
            array_buffer[87] := TO_BYTE(     TO_DWORD(buf5.AnalogSensor.Sensor[5].MIN_VOLT));

            array_buffer[88] := TO_BYTE(SHR(TO_DWORD(buf5.AnalogSensor.Sensor[5].MAX_VOLT),  UINT#24));
            array_buffer[89] := TO_BYTE(SHR(TO_DWORD(buf5.AnalogSensor.Sensor[5].MAX_VOLT),  UINT#16));
            array_buffer[90] := TO_BYTE(SHR(TO_DWORD(buf5.AnalogSensor.Sensor[5].MAX_VOLT),   UINT#8));
            array_buffer[91] := TO_BYTE(     TO_DWORD(buf5.AnalogSensor.Sensor[5].MAX_VOLT));

            array_buffer[92] := TO_BYTE(SHR(TO_DWORD(buf5.AnalogSensor.Sensor[5].MIN_VAL),   UINT#24));
            array_buffer[93] := TO_BYTE(SHR(TO_DWORD(buf5.AnalogSensor.Sensor[5].MIN_VAL),   UINT#16));
            array_buffer[94] := TO_BYTE(SHR(TO_DWORD(buf5.AnalogSensor.Sensor[5].MIN_VAL),    UINT#8));
            array_buffer[95] := TO_BYTE(     TO_DWORD(buf5.AnalogSensor.Sensor[5].MIN_VAL));

            array_buffer[96] := TO_BYTE(SHR(TO_DWORD(buf5.AnalogSensor.Sensor[5].MAX_VAL),   UINT#24));
            array_buffer[97] := TO_BYTE(SHR(TO_DWORD(buf5.AnalogSensor.Sensor[5].MAX_VAL),   UINT#16));
            array_buffer[98] := TO_BYTE(SHR(TO_DWORD(buf5.AnalogSensor.Sensor[5].MAX_VAL),    UINT#8));
            array_buffer[99] := TO_BYTE(     TO_DWORD(buf5.AnalogSensor.Sensor[5].MAX_VAL));

            // --- Sensor[6] (bytes 100..119) ---
            array_buffer[100] := TO_BYTE(SHR(TO_DWORD(buf5.AnalogSensor.Sensor[6].Enable),   UINT#24));
            array_buffer[101] := TO_BYTE(SHR(TO_DWORD(buf5.AnalogSensor.Sensor[6].Enable),   UINT#16));
            array_buffer[102] := TO_BYTE(SHR(TO_DWORD(buf5.AnalogSensor.Sensor[6].Enable),    UINT#8));
            array_buffer[103] := TO_BYTE(     TO_DWORD(buf5.AnalogSensor.Sensor[6].Enable));

            array_buffer[104] := TO_BYTE(SHR(TO_DWORD(buf5.AnalogSensor.Sensor[6].MIN_VOLT), UINT#24));
            array_buffer[105] := TO_BYTE(SHR(TO_DWORD(buf5.AnalogSensor.Sensor[6].MIN_VOLT), UINT#16));
            array_buffer[106] := TO_BYTE(SHR(TO_DWORD(buf5.AnalogSensor.Sensor[6].MIN_VOLT),  UINT#8));
            array_buffer[107] := TO_BYTE(     TO_DWORD(buf5.AnalogSensor.Sensor[6].MIN_VOLT));

            array_buffer[108] := TO_BYTE(SHR(TO_DWORD(buf5.AnalogSensor.Sensor[6].MAX_VOLT), UINT#24));
            array_buffer[109] := TO_BYTE(SHR(TO_DWORD(buf5.AnalogSensor.Sensor[6].MAX_VOLT), UINT#16));
            array_buffer[110] := TO_BYTE(SHR(TO_DWORD(buf5.AnalogSensor.Sensor[6].MAX_VOLT),  UINT#8));
            array_buffer[111] := TO_BYTE(     TO_DWORD(buf5.AnalogSensor.Sensor[6].MAX_VOLT));

            array_buffer[112] := TO_BYTE(SHR(TO_DWORD(buf5.AnalogSensor.Sensor[6].MIN_VAL),  UINT#24));
            array_buffer[113] := TO_BYTE(SHR(TO_DWORD(buf5.AnalogSensor.Sensor[6].MIN_VAL),  UINT#16));
            array_buffer[114] := TO_BYTE(SHR(TO_DWORD(buf5.AnalogSensor.Sensor[6].MIN_VAL),   UINT#8));
            array_buffer[115] := TO_BYTE(     TO_DWORD(buf5.AnalogSensor.Sensor[6].MIN_VAL));

            array_buffer[116] := TO_BYTE(SHR(TO_DWORD(buf5.AnalogSensor.Sensor[6].MAX_VAL),  UINT#24));
            array_buffer[117] := TO_BYTE(SHR(TO_DWORD(buf5.AnalogSensor.Sensor[6].MAX_VAL),  UINT#16));
            array_buffer[118] := TO_BYTE(SHR(TO_DWORD(buf5.AnalogSensor.Sensor[6].MAX_VAL),   UINT#8));
            array_buffer[119] := TO_BYTE(     TO_DWORD(buf5.AnalogSensor.Sensor[6].MAX_VAL));

            // --- Sensor[7] (bytes 120..139) ---
            array_buffer[120] := TO_BYTE(SHR(TO_DWORD(buf5.AnalogSensor.Sensor[7].Enable),   UINT#24));
            array_buffer[121] := TO_BYTE(SHR(TO_DWORD(buf5.AnalogSensor.Sensor[7].Enable),   UINT#16));
            array_buffer[122] := TO_BYTE(SHR(TO_DWORD(buf5.AnalogSensor.Sensor[7].Enable),    UINT#8));
            array_buffer[123] := TO_BYTE(     TO_DWORD(buf5.AnalogSensor.Sensor[7].Enable));

            array_buffer[124] := TO_BYTE(SHR(TO_DWORD(buf5.AnalogSensor.Sensor[7].MIN_VOLT), UINT#24));
            array_buffer[125] := TO_BYTE(SHR(TO_DWORD(buf5.AnalogSensor.Sensor[7].MIN_VOLT), UINT#16));
            array_buffer[126] := TO_BYTE(SHR(TO_DWORD(buf5.AnalogSensor.Sensor[7].MIN_VOLT),  UINT#8));
            array_buffer[127] := TO_BYTE(     TO_DWORD(buf5.AnalogSensor.Sensor[7].MIN_VOLT));

            array_buffer[128] := TO_BYTE(SHR(TO_DWORD(buf5.AnalogSensor.Sensor[7].MAX_VOLT), UINT#24));
            array_buffer[129] := TO_BYTE(SHR(TO_DWORD(buf5.AnalogSensor.Sensor[7].MAX_VOLT), UINT#16));
            array_buffer[130] := TO_BYTE(SHR(TO_DWORD(buf5.AnalogSensor.Sensor[7].MAX_VOLT),  UINT#8));
            array_buffer[131] := TO_BYTE(     TO_DWORD(buf5.AnalogSensor.Sensor[7].MAX_VOLT));

            array_buffer[132] := TO_BYTE(SHR(TO_DWORD(buf5.AnalogSensor.Sensor[7].MIN_VAL),  UINT#24));
            array_buffer[133] := TO_BYTE(SHR(TO_DWORD(buf5.AnalogSensor.Sensor[7].MIN_VAL),  UINT#16));
            array_buffer[134] := TO_BYTE(SHR(TO_DWORD(buf5.AnalogSensor.Sensor[7].MIN_VAL),   UINT#8));
            array_buffer[135] := TO_BYTE(     TO_DWORD(buf5.AnalogSensor.Sensor[7].MIN_VAL));

            array_buffer[136] := TO_BYTE(SHR(TO_DWORD(buf5.AnalogSensor.Sensor[7].MAX_VAL),  UINT#24));
            array_buffer[137] := TO_BYTE(SHR(TO_DWORD(buf5.AnalogSensor.Sensor[7].MAX_VAL),  UINT#16));
            array_buffer[138] := TO_BYTE(SHR(TO_DWORD(buf5.AnalogSensor.Sensor[7].MAX_VAL),   UINT#8));
            array_buffer[139] := TO_BYTE(     TO_DWORD(buf5.AnalogSensor.Sensor[7].MAX_VAL));

            // --- Sensor[8] (bytes 140..159) ---
            array_buffer[140] := TO_BYTE(SHR(TO_DWORD(buf5.AnalogSensor.Sensor[8].Enable),   UINT#24));
            array_buffer[141] := TO_BYTE(SHR(TO_DWORD(buf5.AnalogSensor.Sensor[8].Enable),   UINT#16));
            array_buffer[142] := TO_BYTE(SHR(TO_DWORD(buf5.AnalogSensor.Sensor[8].Enable),    UINT#8));
            array_buffer[143] := TO_BYTE(     TO_DWORD(buf5.AnalogSensor.Sensor[8].Enable));

            array_buffer[144] := TO_BYTE(SHR(TO_DWORD(buf5.AnalogSensor.Sensor[8].MIN_VOLT), UINT#24));
            array_buffer[145] := TO_BYTE(SHR(TO_DWORD(buf5.AnalogSensor.Sensor[8].MIN_VOLT), UINT#16));
            array_buffer[146] := TO_BYTE(SHR(TO_DWORD(buf5.AnalogSensor.Sensor[8].MIN_VOLT),  UINT#8));
            array_buffer[147] := TO_BYTE(     TO_DWORD(buf5.AnalogSensor.Sensor[8].MIN_VOLT));

            array_buffer[148] := TO_BYTE(SHR(TO_DWORD(buf5.AnalogSensor.Sensor[8].MAX_VOLT), UINT#24));
            array_buffer[149] := TO_BYTE(SHR(TO_DWORD(buf5.AnalogSensor.Sensor[8].MAX_VOLT), UINT#16));
            array_buffer[150] := TO_BYTE(SHR(TO_DWORD(buf5.AnalogSensor.Sensor[8].MAX_VOLT),  UINT#8));
            array_buffer[151] := TO_BYTE(     TO_DWORD(buf5.AnalogSensor.Sensor[8].MAX_VOLT));

            array_buffer[152] := TO_BYTE(SHR(TO_DWORD(buf5.AnalogSensor.Sensor[8].MIN_VAL),  UINT#24));
            array_buffer[153] := TO_BYTE(SHR(TO_DWORD(buf5.AnalogSensor.Sensor[8].MIN_VAL),  UINT#16));
            array_buffer[154] := TO_BYTE(SHR(TO_DWORD(buf5.AnalogSensor.Sensor[8].MIN_VAL),   UINT#8));
            array_buffer[155] := TO_BYTE(     TO_DWORD(buf5.AnalogSensor.Sensor[8].MIN_VAL));

            array_buffer[156] := TO_BYTE(SHR(TO_DWORD(buf5.AnalogSensor.Sensor[8].MAX_VAL),  UINT#24));
            array_buffer[157] := TO_BYTE(SHR(TO_DWORD(buf5.AnalogSensor.Sensor[8].MAX_VAL),  UINT#16));
            array_buffer[158] := TO_BYTE(SHR(TO_DWORD(buf5.AnalogSensor.Sensor[8].MAX_VAL),   UINT#8));
            array_buffer[159] := TO_BYTE(     TO_DWORD(buf5.AnalogSensor.Sensor[8].MAX_VAL));

            // --- AfterburstEnable (bytes 160..163) ---
            array_buffer[160] := TO_BYTE(SHR(TO_DWORD(buf5.AfterburstEnable), UINT#24));
            array_buffer[161] := TO_BYTE(SHR(TO_DWORD(buf5.AfterburstEnable), UINT#16));
            array_buffer[162] := TO_BYTE(SHR(TO_DWORD(buf5.AfterburstEnable),  UINT#8));
            array_buffer[163] := TO_BYTE(     TO_DWORD(buf5.AfterburstEnable));

            // --- LimitWeld1TimeEnable bits (bytes 164..167) ---
            array_buffer[164].%X0 := buf5.LimitWeld1TimeEnable._0;
            array_buffer[164].%X1 := buf5.LimitWeld1TimeEnable._1;
            array_buffer[164].%X2 := buf5.LimitWeld1TimeEnable._2;
            array_buffer[164].%X3 := buf5.LimitWeld1TimeEnable._3;
            array_buffer[164].%X4 := buf5.LimitWeld1TimeEnable._4;
            array_buffer[164].%X5 := buf5.LimitWeld1TimeEnable._5;
            array_buffer[164].%X6 := buf5.LimitWeld1TimeEnable._6;
            array_buffer[164].%X7 := buf5.LimitWeld1TimeEnable._7;

            array_buffer[165].%X0 := buf5.LimitWeld1TimeEnable._8;
            array_buffer[165].%X1 := buf5.LimitWeld1TimeEnable._9;
            array_buffer[165].%X2 := buf5.LimitWeld1TimeEnable._10;
            array_buffer[165].%X3 := buf5.LimitWeld1TimeEnable._11;
            array_buffer[165].%X4 := buf5.LimitWeld1TimeEnable._12;
            array_buffer[165].%X5 := buf5.LimitWeld1TimeEnable._13;
            array_buffer[165].%X6 := buf5.LimitWeld1TimeEnable._14;
            array_buffer[165].%X7 := buf5.LimitWeld1TimeEnable._15;

            array_buffer[166].%X0 := buf5.LimitWeld1TimeEnable._16;
            array_buffer[166].%X1 := buf5.LimitWeld1TimeEnable._17;
            array_buffer[166].%X2 := buf5.LimitWeld1TimeEnable._18;
            array_buffer[166].%X3 := buf5.LimitWeld1TimeEnable._19;
            array_buffer[166].%X4 := buf5.LimitWeld1TimeEnable._20;
            array_buffer[166].%X5 := buf5.LimitWeld1TimeEnable._21;
            array_buffer[166].%X6 := buf5.LimitWeld1TimeEnable._22;
            array_buffer[166].%X7 := buf5.LimitWeld1TimeEnable._23;

            array_buffer[167].%X0 := buf5.LimitWeld1TimeEnable.LowerBad_1;
            array_buffer[167].%X1 := buf5.LimitWeld1TimeEnable.LowerSuspect_1;
            array_buffer[167].%X2 := buf5.LimitWeld1TimeEnable.UpperSuspect_1;
            array_buffer[167].%X3 := buf5.LimitWeld1TimeEnable.UpperBad_1;
            array_buffer[167].%X4 := buf5.LimitWeld1TimeEnable.Display_1;
            array_buffer[167].%X5 := buf5.LimitWeld1TimeEnable._29;
            array_buffer[167].%X6 := buf5.LimitWeld1TimeEnable._30;
            array_buffer[167].%X7 := buf5.LimitWeld1TimeEnable._31;

            // --- LimitWeld1EnergyEnable bits (bytes 168..171) ---
            array_buffer[168].%X0 := buf5.LimitWeld1EnergyEnable._0;
            array_buffer[168].%X1 := buf5.LimitWeld1EnergyEnable._1;
            array_buffer[168].%X2 := buf5.LimitWeld1EnergyEnable._2;
            array_buffer[168].%X3 := buf5.LimitWeld1EnergyEnable._3;
            array_buffer[168].%X4 := buf5.LimitWeld1EnergyEnable._4;
            array_buffer[168].%X5 := buf5.LimitWeld1EnergyEnable._5;
            array_buffer[168].%X6 := buf5.LimitWeld1EnergyEnable._6;
            array_buffer[168].%X7 := buf5.LimitWeld1EnergyEnable._7;
